   S708_TL_DC_U262_1_UP_DN.Error_T1.STATE := B#16#0;
   S708_TL_DC_U262_1_UP_DN.Error_T1.STIME := T#23D5H8M46S781MS;
   S708_TL_DC_U262_1_UP_DN.Error_T1.ATIME := T#23D5H8M46S825MS;
   S708_TL_DC_U262_1_UP_DN.Error_T2.IN := FALSE;
   S708_TL_DC_U262_1_UP_DN.Error_T2.PT := T#4S;
   S708_TL_DC_U262_1_UP_DN.Error_T2.Q := FALSE;
   S708_TL_DC_U262_1_UP_DN.Error_T2.ET := T#0MS;
   S708_TL_DC_U262_1_UP_DN.Error_T2.STATE := B#16#0;
   S708_TL_DC_U262_1_UP_DN.Error_T2.STIME := T#0MS;
   S708_TL_DC_U262_1_UP_DN.Error_T2.ATIME := T#0MS;
   S708_TL_DC_U262_1_UP_DN.Adv_End_Aux := FALSE;
   S708_TL_DC_U262_1_UP_DN.Ret_End_Aux := FALSE;
   S708_TL_DC_U262_1_UP_DN.CHK_Aux1 := FALSE;
   S708_TL_DC_U262_1_UP_DN.CHK_Aux2 := FALSE;
   S708_TL_DC_U262_1_UP_DN.Error_T1_DN := FALSE;
   S708_TL_DC_U262_1_UP_DN.Error_T2_DN := FALSE;
   S708_TL_DC_U262_1_UP_DN.Adv_Memo := FALSE;
   S708_TL_DC_U262_1_UP_DN.Visu_Adv_Arr[0] := FALSE;
   S708_TL_DC_U262_1_UP_DN.Visu_Adv_Arr[1] := FALSE;
   S708_TL_DC_U262_1_UP_DN.Visu_Adv_Arr[2] := FALSE;
   S708_TL_DC_U262_1_UP_DN.Visu_Adv_Arr[3] := FALSE;
   S708_TL_DC_U262_1_UP_DN.Visu_Adv_Arr[4] := FALSE;
   S708_TL_DC_U262_1_UP_DN.Visu_Adv_Arr[5] := FALSE;
   S708_TL_DC_U262_1_UP_DN.Visu_Adv_Arr[6] := FALSE;
   S708_TL_DC_U262_1_UP_DN.Visu_Adv_Arr[7] := FALSE;
   S708_TL_DC_U262_1_UP_DN.Visu_Adv_Arr[8] := FALSE;
   S708_TL_DC_U262_1_UP_DN.Visu_Adv_Arr[9] := FALSE;
   S708_TL_DC_U262_1_UP_DN.Visu_Adv_Arr[10] := FALSE;
   S708_TL_DC_U262_1_UP_DN.Visu_Adv_Arr[11] := FALSE;
   S708_TL_DC_U262_1_UP_DN.Visu_Adv_Arr[12] := FALSE;
   S708_TL_DC_U262_1_UP_DN.Visu_Adv_Arr[13] := FALSE;
   S708_TL_DC_U262_1_UP_DN.Visu_Adv_Arr[14] := FALSE;
   S708_TL_DC_U262_1_UP_DN.Visu_Adv_Arr[15] := FALSE;
   S708_TL_DC_U262_1_UP_DN.Visu_Ret_Arr[0] := FALSE;
   S708_TL_DC_U262_1_UP_DN.Visu_Ret_Arr[1] := FALSE;
   S708_TL_DC_U262_1_UP_DN.Visu_Ret_Arr[2] := FALSE;
   S708_TL_DC_U262_1_UP_DN.Visu_Ret_Arr[3] := FALSE;
   S708_TL_DC_U262_1_UP_DN.Visu_Ret_Arr[4] := FALSE;
   S708_TL_DC_U262_1_UP_DN.Visu_Ret_Arr[5] := FALSE;
   S708_TL_DC_U262_1_UP_DN.Visu_Ret_Arr[6] := FALSE;
   S708_TL_DC_U262_1_UP_DN.Visu_Ret_Arr[7] := FALSE;
   S708_TL_DC_U262_1_UP_DN.Visu_Ret_Arr[8] := FALSE;
   S708_TL_DC_U262_1_UP_DN.Visu_Ret_Arr[9] := FALSE;
   S708_TL_DC_U262_1_UP_DN.Visu_Ret_Arr[10] := FALSE;
   S708_TL_DC_U262_1_UP_DN.Visu_Ret_Arr[11] := FALSE;
   S708_TL_DC_U262_1_UP_DN.Visu_Ret_Arr[12] := FALSE;
   S708_TL_DC_U262_1_UP_DN.Visu_Ret_Arr[13] := FALSE;
   S708_TL_DC_U262_1_UP_DN.Visu_Ret_Arr[14] := FALSE;
   S708_TL_DC_U262_1_UP_DN.Visu_Ret_Arr[15] := FALSE;
   S708_TL_DC_U262_1_UP_DN.BLK_Move_Ret := 0;
   S708_TL_DC_U262_1_UP_DN.Enable := FALSE;
   S708_TL_DC_U262_1_UP_DN.Adv_End := FALSE;
   S708_TL_DC_U262_1_UP_DN.Ret_End := FALSE;
   S708_TL_DC_U262_1.Enable_Aux := FALSE;
   S708_TL_DC_U262_1.Adv_Amount := 1;
   S708_TL_DC_U262_1.Ret_Amount := 1;
   S708_TL_DC_U262_1.LS_Adv1 := FALSE;
   S708_TL_DC_U262_1.LS_Ret1 := FALSE;
   S708_TL_DC_U262_1.LS_Adv2 := FALSE;
   S708_TL_DC_U262_1.LS_Ret2 := FALSE;
   S708_TL_DC_U262_1.LS_Adv3 := FALSE;
   S708_TL_DC_U262_1.LS_Ret3 := FALSE;
   S708_TL_DC_U262_1.LS_Adv4 := FALSE;
   S708_TL_DC_U262_1.LS_Ret4 := FALSE;
   S708_TL_DC_U262_1.LS_Adv5 := FALSE;
   S708_TL_DC_U262_1.LS_Ret5 := FALSE;
   S708_TL_DC_U262_1.LS_Adv6 := FALSE;
   S708_TL_DC_U262_1.LS_Ret6 := FALSE;
   S708_TL_DC_U262_1.LS_Adv7 := FALSE;
   S708_TL_DC_U262_1.LS_Ret7 := FALSE;
   S708_TL_DC_U262_1.LS_Adv8 := FALSE;
   S708_TL_DC_U262_1.LS_Ret8 := FALSE;
   S708_TL_DC_U262_1.SOL_Adv := FALSE;
   S708_TL_DC_U262_1.SOL_Ret := FALSE;
   S708_TL_DC_U262_1.M_Ready := TRUE;
   S708_TL_DC_U262_1.T_CHK1 := T#4S;
   S708_TL_DC_U262_1.T_CHK2 := T#4S;
   S708_TL_DC_U262_1.PB_Lamp_CHK := FALSE;
   S708_TL_DC_U262_1.PB_Error_Rst := FALSE;
   S708_TL_DC_U262_1.M_FLICK := TRUE;
   S708_TL_DC_U262_1.M_Adv_Err := FALSE;
   S708_TL_DC_U262_1.M_Ret_Err := FALSE;
   S708_TL_DC_U262_1.LP_Adv := FALSE;
   S708_TL_DC_U262_1.LP_Ret := FALSE;
   S708_TL_DC_U262_1.Visu_Adv := W#16#0;
   S708_TL_DC_U262_1.Visu_Ret := W#16#0;
   S708_TL_DC_U262_1.Error_T1.IN := FALSE;
   S708_TL_DC_U262_1.Error_T1.PT := T#4S;
   S708_TL_DC_U262_1.Error_T1.Q := FALSE;
   S708_TL_DC_U262_1.Error_T1.ET := T#0MS;
   S708_TL_DC_U262_1.Error_T1.STATE := B#16#0;
   S708_TL_DC_U262_1.Error_T1.STIME := T#23D5H8M46S781MS;
   S708_TL_DC_U262_1.Error_T1.ATIME := T#23D5H8M46S825MS;
   S708_TL_DC_U262_1.Error_T2.IN := FALSE;
   S708_TL_DC_U262_1.Error_T2.PT := T#4S;
   S708_TL_DC_U262_1.Error_T2.Q := FALSE;
   S708_TL_DC_U262_1.Error_T2.ET := T#0MS;
   S708_TL_DC_U262_1.Error_T2.STATE := B#16#0;
   S708_TL_DC_U262_1.Error_T2.STIME := T#13H51M46S5MS;
   S708_TL_DC_U262_1.Error_T2.ATIME := T#13H51M46S50MS;
   S708_TL_DC_U262_1.Adv_End_Aux := FALSE;
   S708_TL_DC_U262_1.Ret_End_Aux := FALSE;
   S708_TL_DC_U262_1.CHK_Aux1 := FALSE;
   S708_TL_DC_U262_1.CHK_Aux2 := FALSE;
   S708_TL_DC_U262_1.Error_T1_DN := FALSE;
   S708_TL_DC_U262_1.Error_T2_DN := FALSE;
   S708_TL_DC_U262_1.Adv_Memo := FALSE;
   S708_TL_DC_U262_1.Visu_Adv_Arr[0] := FALSE;
   S708_TL_DC_U262_1.Visu_Adv_Arr[1] := FALSE;
   S708_TL_DC_U262_1.Visu_Adv_Arr[2] := FALSE;
   S708_TL_DC_U262_1.Visu_Adv_Arr[3] := FALSE;
   S708_TL_DC_U262_1.Visu_Adv_Arr[4] := FALSE;
   S708_TL_DC_U262_1.Visu_Adv_Arr[5] := FALSE;
   S708_TL_DC_U262_1.Visu_Adv_Arr[6] := FALSE;
   S708_TL_DC_U262_1.Visu_Adv_Arr[7] := FALSE;
   S708_TL_DC_U262_1.Visu_Adv_Arr[8] := FALSE;
   S708_TL_DC_U262_1.Visu_Adv_Arr[9] := FALSE;
   S708_TL_DC_U262_1.Visu_Adv_Arr[10] := FALSE;
   S708_TL_DC_U262_1.Visu_Adv_Arr[11] := FALSE;
   S708_TL_DC_U262_1.Visu_Adv_Arr[12] := FALSE;
   S708_TL_DC_U262_1.Visu_Adv_Arr[13] := FALSE;
   S708_TL_DC_U262_1.Visu_Adv_Arr[14] := FALSE;
   S708_TL_DC_U262_1.Visu_Adv_Arr[15] := FALSE;
   S708_TL_DC_U262_1.Visu_Ret_Arr[0] := FALSE;
   S708_TL_DC_U262_1.Visu_Ret_Arr[1] := FALSE;
   S708_TL_DC_U262_1.Visu_Ret_Arr[2] := FALSE;
   S708_TL_DC_U262_1.Visu_Ret_Arr[3] := FALSE;
   S708_TL_DC_U262_1.Visu_Ret_Arr[4] := FALSE;
   S708_TL_DC_U262_1.Visu_Ret_Arr[5] := FALSE;
   S708_TL_DC_U262_1.Visu_Ret_Arr[6] := FALSE;
   S708_TL_DC_U262_1.Visu_Ret_Arr[7] := FALSE;
   S708_TL_DC_U262_1.Visu_Ret_Arr[8] := FALSE;
   S708_TL_DC_U262_1.Visu_Ret_Arr[9] := FALSE;
   S708_TL_DC_U262_1.Visu_Ret_Arr[10] := FALSE;
   S708_TL_DC_U262_1.Visu_Ret_Arr[11] := FALSE;
   S708_TL_DC_U262_1.Visu_Ret_Arr[12] := FALSE;
   S708_TL_DC_U262_1.Visu_Ret_Arr[13] := FALSE;
   S708_TL_DC_U262_1.Visu_Ret_Arr[14] := FALSE;
   S708_TL_DC_U262_1.Visu_Ret_Arr[15] := FALSE;
   S708_TL_DC_U262_1.BLK_Move_Ret := 0;
   S708_TL_DC_U262_1.Enable := FALSE;
   S708_TL_DC_U262_1.Adv_End := FALSE;
   S708_TL_DC_U262_1.Ret_End := FALSE;
   S708_TL_DC_U262_1_CLAMP.Enable_Aux := FALSE;
   S708_TL_DC_U262_1_CLAMP.Adv_Amount := 1;
   S708_TL_DC_U262_1_CLAMP.Ret_Amount := 1;
   S708_TL_DC_U262_1_CLAMP.LS_Adv1 := FALSE;
   S708_TL_DC_U262_1_CLAMP.LS_Ret1 := FALSE;
   S708_TL_DC_U262_1_CLAMP.LS_Adv2 := FALSE;
   S708_TL_DC_U262_1_CLAMP.LS_Ret2 := FALSE;
   S708_TL_DC_U262_1_CLAMP.LS_Adv3 := FALSE;
   S708_TL_DC_U262_1_CLAMP.LS_Ret3 := FALSE;
   S708_TL_DC_U262_1_CLAMP.LS_Adv4 := FALSE;
   S708_TL_DC_U262_1_CLAMP.LS_Ret4 := FALSE;
   S708_TL_DC_U262_1_CLAMP.LS_Adv5 := FALSE;
   S708_TL_DC_U262_1_CLAMP.LS_Ret5 := FALSE;
   S708_TL_DC_U262_1_CLAMP.LS_Adv6 := FALSE;
   S708_TL_DC_U262_1_CLAMP.LS_Ret6 := FALSE;
   S708_TL_DC_U262_1_CLAMP.LS_Adv7 := FALSE;
   S708_TL_DC_U262_1_CLAMP.LS_Ret7 := FALSE;
   S708_TL_DC_U262_1_CLAMP.LS_Adv8 := FALSE;
   S708_TL_DC_U262_1_CLAMP.LS_Ret8 := FALSE;
   S708_TL_DC_U262_1_CLAMP.SOL_Adv := FALSE;
   S708_TL_DC_U262_1_CLAMP.SOL_Ret := FALSE;
   S708_TL_DC_U262_1_CLAMP.M_Ready := TRUE;
   S708_TL_DC_U262_1_CLAMP.T_CHK1 := T#4S;
   S708_TL_DC_U262_1_CLAMP.T_CHK2 := T#4S;
   S708_TL_DC_U262_1_CLAMP.PB_Lamp_CHK := FALSE;
   S708_TL_DC_U262_1_CLAMP.PB_Error_Rst := FALSE;
   S708_TL_DC_U262_1_CLAMP.M_FLICK := TRUE;
   S708_TL_DC_U262_1_CLAMP.M_Adv_Err := FALSE;
   S708_TL_DC_U262_1_CLAMP.M_Ret_Err := FALSE;
   S708_TL_DC_U262_1_CLAMP.LP_Adv := FALSE;
   S708_TL_DC_U262_1_CLAMP.LP_Ret := FALSE;
   S708_TL_DC_U262_1_CLAMP.Visu_Adv := W#16#0;
   S708_TL_DC_U262_1_CLAMP.Visu_Ret := W#16#0;
   S708_TL_DC_U262_1_CLAMP.Error_T1.IN := FALSE;
   S708_TL_DC_U262_1_CLAMP.Error_T1.PT := T#4S;
   S708_TL_DC_U262_1_CLAMP.Error_T1.Q := FALSE;
   S708_TL_DC_U262_1_CLAMP.Error_T1.ET := T#0MS;
   S708_TL_DC_U262_1_CLAMP.Error_T1.STATE := B#16#0;
   S708_TL_DC_U262_1_CLAMP.Error_T1.STIME := T#23D5H8M46S781MS;
   S708_TL_DC_U262_1_CLAMP.Error_T1.ATIME := T#23D5H8M46S825MS;
   S708_TL_DC_U262_1_CLAMP.Error_T2.IN := FALSE;
   S708_TL_DC_U262_1_CLAMP.Error_T2.PT := T#4S;
   S708_TL_DC_U262_1_CLAMP.Error_T2.Q := FALSE;
   S708_TL_DC_U262_1_CLAMP.Error_T2.ET := T#0MS;
   S708_TL_DC_U262_1_CLAMP.Error_T2.STATE := B#16#0;
   S708_TL_DC_U262_1_CLAMP.Error_T2.STIME := T#0MS;
   S708_TL_DC_U262_1_CLAMP.Error_T2.ATIME := T#0MS;
   S708_TL_DC_U262_1_CLAMP.Adv_End_Aux := FALSE;
   S708_TL_DC_U262_1_CLAMP.Ret_End_Aux := FALSE;
   S708_TL_DC_U262_1_CLAMP.CHK_Aux1 := FALSE;
   S708_TL_DC_U262_1_CLAMP.CHK_Aux2 := FALSE;
   S708_TL_DC_U262_1_CLAMP.Error_T1_DN := FALSE;
   S708_TL_DC_U262_1_CLAMP.Error_T2_DN := FALSE;
   S708_TL_DC_U262_1_CLAMP.Adv_Memo := FALSE;
   S708_TL_DC_U262_1_CLAMP.Visu_Adv_Arr[0] := FALSE;
   S708_TL_DC_U262_1_CLAMP.Visu_Adv_Arr[1] := FALSE;
   S708_TL_DC_U262_1_CLAMP.Visu_Adv_Arr[2] := FALSE;
   S708_TL_DC_U262_1_CLAMP.Visu_Adv_Arr[3] := FALSE;
   S708_TL_DC_U262_1_CLAMP.Visu_Adv_Arr[4] := FALSE;
   S708_TL_DC_U262_1_CLAMP.Visu_Adv_Arr[5] := FALSE;
   S708_TL_DC_U262_1_CLAMP.Visu_Adv_Arr[6] := FALSE;
   S708_TL_DC_U262_1_CLAMP.Visu_Adv_Arr[7] := FALSE;
   S708_TL_DC_U262_1_CLAMP.Visu_Adv_Arr[8] := FALSE;
   S708_TL_DC_U262_1_CLAMP.Visu_Adv_Arr[9] := FALSE;
   S708_TL_DC_U262_1_CLAMP.Visu_Adv_Arr[10] := FALSE;
   S708_TL_DC_U262_1_CLAMP.Visu_Adv_Arr[11] := FALSE;
   S708_TL_DC_U262_1_CLAMP.Visu_Adv_Arr[12] := FALSE;
   S708_TL_DC_U262_1_CLAMP.Visu_Adv_Arr[13] := FALSE;
   S708_TL_DC_U262_1_CLAMP.Visu_Adv_Arr[14] := FALSE;
   S708_TL_DC_U262_1_CLAMP.Visu_Adv_Arr[15] := FALSE;
   S708_TL_DC_U262_1_CLAMP.Visu_Ret_Arr[0] := FALSE;
   S708_TL_DC_U262_1_CLAMP.Visu_Ret_Arr[1] := FALSE;
   S708_TL_DC_U262_1_CLAMP.Visu_Ret_Arr[2] := FALSE;
   S708_TL_DC_U262_1_CLAMP.Visu_Ret_Arr[3] := FALSE;
   S708_TL_DC_U262_1_CLAMP.Visu_Ret_Arr[4] := FALSE;
   S708_TL_DC_U262_1_CLAMP.Visu_Ret_Arr[5] := FALSE;
   S708_TL_DC_U262_1_CLAMP.Visu_Ret_Arr[6] := FALSE;
   S708_TL_DC_U262_1_CLAMP.Visu_Ret_Arr[7] := FALSE;
   S708_TL_DC_U262_1_CLAMP.Visu_Ret_Arr[8] := FALSE;
   S708_TL_DC_U262_1_CLAMP.Visu_Ret_Arr[9] := FALSE;
   S708_TL_DC_U262_1_CLAMP.Visu_Ret_Arr[10] := FALSE;
   S708_TL_DC_U262_1_CLAMP.Visu_Ret_Arr[11] := FALSE;
   S708_TL_DC_U262_1_CLAMP.Visu_Ret_Arr[12] := FALSE;
   S708_TL_DC_U262_1_CLAMP.Visu_Ret_Arr[13] := FALSE;
   S708_TL_DC_U262_1_CLAMP.Visu_Ret_Arr[14] := FALSE;
   S708_TL_DC_U262_1_CLAMP.Visu_Ret_Arr[15] := FALSE;
   S708_TL_DC_U262_1_CLAMP.BLK_Move_Ret := 0;
   S708_TL_DC_U262_1_CLAMP.Enable := FALSE;
   S708_TL_DC_U262_1_CLAMP.Adv_End := FALSE;
   S708_TL_DC_U262_1_CLAMP.Ret_End := FALSE;
   S708_TL_DC_U261_2_CLAMP.Enable_Aux := FALSE;
   S708_TL_DC_U261_2_CLAMP.Adv_Amount := 1;
   S708_TL_DC_U261_2_CLAMP.Ret_Amount := 1;
   S708_TL_DC_U261_2_CLAMP.LS_Adv1 := FALSE;
   S708_TL_DC_U261_2_CLAMP.LS_Ret1 := FALSE;
   S708_TL_DC_U261_2_CLAMP.LS_Adv2 := FALSE;
   S708_TL_DC_U261_2_CLAMP.LS_Ret2 := FALSE;
   S708_TL_DC_U261_2_CLAMP.LS_Adv3 := FALSE;
   S708_TL_DC_U261_2_CLAMP.LS_Ret3 := FALSE;
   S708_TL_DC_U261_2_CLAMP.LS_Adv4 := FALSE;
   S708_TL_DC_U261_2_CLAMP.LS_Ret4 := FALSE;
   S708_TL_DC_U261_2_CLAMP.LS_Adv5 := FALSE;
   S708_TL_DC_U261_2_CLAMP.LS_Ret5 := FALSE;
   S708_TL_DC_U261_2_CLAMP.LS_Adv6 := FALSE;
   S708_TL_DC_U261_2_CLAMP.LS_Ret6 := FALSE;
   S708_TL_DC_U261_2_CLAMP.LS_Adv7 := FALSE;
   S708_TL_DC_U261_2_CLAMP.LS_Ret7 := FALSE;
   S708_TL_DC_U261_2_CLAMP.LS_Adv8 := FALSE;
   S708_TL_DC_U261_2_CLAMP.LS_Ret8 := FALSE;
   S708_TL_DC_U261_2_CLAMP.SOL_Adv := FALSE;
   S708_TL_DC_U261_2_CLAMP.SOL_Ret := FALSE;
   S708_TL_DC_U261_2_CLAMP.M_Ready := TRUE;
   S708_TL_DC_U261_2_CLAMP.T_CHK1 := T#4S;
   S708_TL_DC_U261_2_CLAMP.T_CHK2 := T#4S;
   S708_TL_DC_U261_2_CLAMP.PB_Lamp_CHK := FALSE;
   S708_TL_DC_U261_2_CLAMP.PB_Error_Rst := FALSE;
   S708_TL_DC_U261_2_CLAMP.M_FLICK := TRUE;
   S708_TL_DC_U261_2_CLAMP.M_Adv_Err := FALSE;
   S708_TL_DC_U261_2_CLAMP.M_Ret_Err := FALSE;
   S708_TL_DC_U261_2_CLAMP.LP_Adv := FALSE;
   S708_TL_DC_U261_2_CLAMP.LP_Ret := FALSE;
   S708_TL_DC_U261_2_CLAMP.Visu_Adv := W#16#0;
   S708_TL_DC_U261_2_CLAMP.Visu_Ret := W#16#0;
   S708_TL_DC_U261_2_CLAMP.Error_T1.IN := FALSE;
   S708_TL_DC_U261_2_CLAMP.Error_T1.PT := T#4S;
   S708_TL_DC_U261_2_CLAMP.Error_T1.Q := FALSE;
   S708_TL_DC_U261_2_CLAMP.Error_T1.ET := T#0MS;
   S708_TL_DC_U261_2_CLAMP.Error_T1.STATE := B#16#0;
   S708_TL_DC_U261_2_CLAMP.Error_T1.STIME := T#23D5H8M46S781MS;
   S708_TL_DC_U261_2_CLAMP.Error_T1.ATIME := T#23D5H8M46S825MS;
   S708_TL_DC_U261_2_CLAMP.Error_T2.IN := FALSE;
   S708_TL_DC_U261_2_CLAMP.Error_T2.PT := T#4S;
   S708_TL_DC_U261_2_CLAMP.Error_T2.Q := FALSE;
   S708_TL_DC_U261_2_CLAMP.Error_T2.ET := T#0MS;
   S708_TL_DC_U261_2_CLAMP.Error_T2.STATE := B#16#0;
   S708_TL_DC_U261_2_CLAMP.Error_T2.STIME := T#0MS;
   S708_TL_DC_U261_2_CLAMP.Error_T2.ATIME := T#0MS;
   S708_TL_DC_U261_2_CLAMP.Adv_End_Aux := FALSE;
   S708_TL_DC_U261_2_CLAMP.Ret_End_Aux := FALSE;
   S708_TL_DC_U261_2_CLAMP.CHK_Aux1 := FALSE;
   S708_TL_DC_U261_2_CLAMP.CHK_Aux2 := FALSE;
   S708_TL_DC_U261_2_CLAMP.Error_T1_DN := FALSE;
   S708_TL_DC_U261_2_CLAMP.Error_T2_DN := FALSE;
   S708_TL_DC_U261_2_CLAMP.Adv_Memo := FALSE;
   S708_TL_DC_U261_2_CLAMP.Visu_Adv_Arr[0] := FALSE;
   S708_TL_DC_U261_2_CLAMP.Visu_Adv_Arr[1] := FALSE;
   S708_TL_DC_U261_2_CLAMP.Visu_Adv_Arr[2] := FALSE;
   S708_TL_DC_U261_2_CLAMP.Visu_Adv_Arr[3] := FALSE;
   S708_TL_DC_U261_2_CLAMP.Visu_Adv_Arr[4] := FALSE;
   S708_TL_DC_U261_2_CLAMP.Visu_Adv_Arr[5] := FALSE;
   S708_TL_DC_U261_2_CLAMP.Visu_Adv_Arr[6] := FALSE;
   S708_TL_DC_U261_2_CLAMP.Visu_Adv_Arr[7] := FALSE;
   S708_TL_DC_U261_2_CLAMP.Visu_Adv_Arr[8] := FALSE;
   S708_TL_DC_U261_2_CLAMP.Visu_Adv_Arr[9] := FALSE;
   S708_TL_DC_U261_2_CLAMP.Visu_Adv_Arr[10] := FALSE;
   S708_TL_DC_U261_2_CLAMP.Visu_Adv_Arr[11] := FALSE;
   S708_TL_DC_U261_2_CLAMP.Visu_Adv_Arr[12] := FALSE;
   S708_TL_DC_U261_2_CLAMP.Visu_Adv_Arr[13] := FALSE;
   S708_TL_DC_U261_2_CLAMP.Visu_Adv_Arr[14] := FALSE;
   S708_TL_DC_U261_2_CLAMP.Visu_Adv_Arr[15] := FALSE;
   S708_TL_DC_U261_2_CLAMP.Visu_Ret_Arr[0] := FALSE;
   S708_TL_DC_U261_2_CLAMP.Visu_Ret_Arr[1] := FALSE;
   S708_TL_DC_U261_2_CLAMP.Visu_Ret_Arr[2] := FALSE;
   S708_TL_DC_U261_2_CLAMP.Visu_Ret_Arr[3] := FALSE;
   S708_TL_DC_U261_2_CLAMP.Visu_Ret_Arr[4] := FALSE;
   S708_TL_DC_U261_2_CLAMP.Visu_Ret_Arr[5] := FALSE;
   S708_TL_DC_U261_2_CLAMP.Visu_Ret_Arr[6] := FALSE;
   S708_TL_DC_U261_2_CLAMP.Visu_Ret_Arr[7] := FALSE;
   S708_TL_DC_U261_2_CLAMP.Visu_Ret_Arr[8] := FALSE;
   S708_TL_DC_U261_2_CLAMP.Visu_Ret_Arr[9] := FALSE;
   S708_TL_DC_U261_2_CLAMP.Visu_Ret_Arr[10] := FALSE;
   S708_TL_DC_U261_2_CLAMP.Visu_Ret_Arr[11] := FALSE;
   S708_TL_DC_U261_2_CLAMP.Visu_Ret_Arr[12] := FALSE;
   S708_TL_DC_U261_2_CLAMP.Visu_Ret_Arr[13] := FALSE;
   S708_TL_DC_U261_2_CLAMP.Visu_Ret_Arr[14] := FALSE;
   S708_TL_DC_U261_2_CLAMP.Visu_Ret_Arr[15] := FALSE;
   S708_TL_DC_U261_2_CLAMP.BLK_Move_Ret := 0;
   S708_TL_DC_U261_2_CLAMP.Enable := FALSE;
   S708_TL_DC_U261_2_CLAMP.Adv_End := FALSE;
   S708_TL_DC_U261_2_CLAMP.Ret_End := FALSE;
END_DATA_BLOCK

FUNCTION FC 144 : VOID
TITLE =
VERSION : 0.1

BEGIN
NETWORK
TITLE =
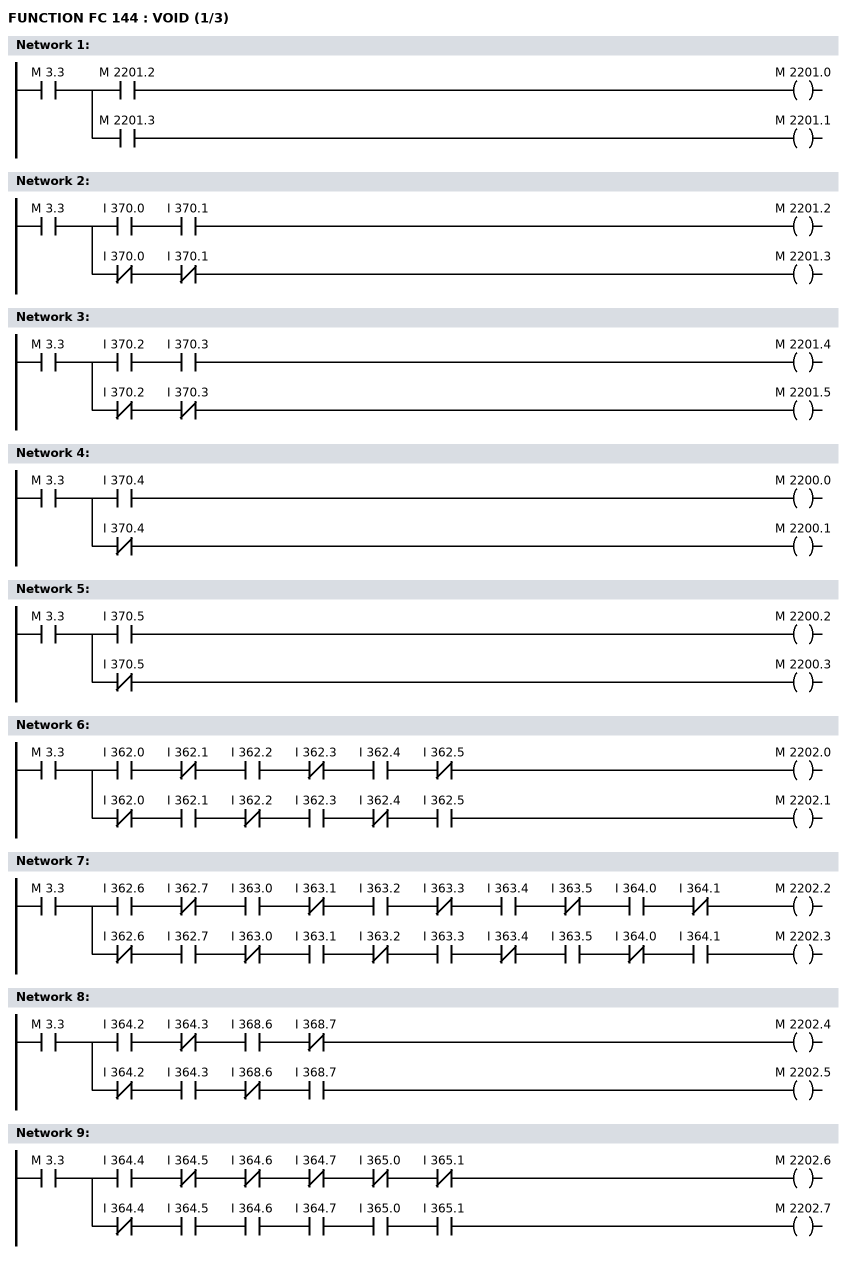

      A     M      3.3;
      =     L      0.0;
      A     L      0.0;
      A     M   2201.2;
      =     M   2201.0;
      A     L      0.0;
      A     M   2201.3;
      =     M   2201.1;
NETWORK
TITLE =

      A     M      3.3;
      =     L      0.0;
      A     L      0.0;
      A     I    370.0;
      A     I    370.1;
      =     M   2201.2;
      A     L      0.0;
      AN    I    370.0;
      AN    I    370.1;
      =     M   2201.3;
NETWORK
TITLE =

      A     M      3.3;
      =     L      0.0;
      A     L      0.0;
      A     I    370.2;
      A     I    370.3;
      =     M   2201.4;
      A     L      0.0;
      AN    I    370.2;
      AN    I    370.3;
      =     M   2201.5;
NETWORK
TITLE =

      A     M      3.3;
      =     L      0.0;
      A     L      0.0;
      A     I    370.4;
      =     M   2200.0;
      A     L      0.0;
      AN    I    370.4;
      =     M   2200.1;
NETWORK
TITLE =

      A     M      3.3;
      =     L      0.0;
      A     L      0.0;
      A     I    370.5;
      =     M   2200.2;
      A     L      0.0;
      AN    I    370.5;
      =     M   2200.3;
NETWORK
TITLE =

      A     M      3.3;
      =     L      0.0;
      A     L      0.0;
      A     I    362.0;
      AN    I    362.1;
      A     I    362.2;
      AN    I    362.3;
      A     I    362.4;
      AN    I    362.5;
      =     M   2202.0;
      A     L      0.0;
      AN    I    362.0;
      A     I    362.1;
      AN    I    362.2;
      A     I    362.3;
      AN    I    362.4;
      A     I    362.5;
      =     M   2202.1;
NETWORK
TITLE =

      A     M      3.3;
      =     L      0.0;
      A     L      0.0;
      A     I    362.6;
      AN    I    362.7;
      A     I    363.0;
      AN    I    363.1;
      A     I    363.2;
      AN    I    363.3;
      A     I    363.4;
      AN    I    363.5;
      A     I    364.0;
      AN    I    364.1;
      =     M   2202.2;
      A     L      0.0;
      AN    I    362.6;
      A     I    362.7;
      AN    I    363.0;
      A     I    363.1;
      AN    I    363.2;
      A     I    363.3;
      AN    I    363.4;
      A     I    363.5;
      AN    I    364.0;
      A     I    364.1;
      =     M   2202.3;
NETWORK
TITLE =

      A     M      3.3;
      =     L      0.0;
      A     L      0.0;
      A     I    364.2;
      AN    I    364.3;
      A     I    368.6;
      AN    I    368.7;
      =     M   2202.4;
      A     L      0.0;
      AN    I    364.2;
      A     I    364.3;
      AN    I    368.6;
      A     I    368.7;
      =     M   2202.5;
NETWORK
TITLE =

      A     M      3.3;
      =     L      0.0;
      A     L      0.0;
      A     I    364.4;
      AN    I    364.5;
      AN    I    364.6;
      AN    I    364.7;
      AN    I    365.0;
      AN    I    365.1;
      =     M   2202.6;
      A     L      0.0;
      AN    I    364.4;
      A     I    364.5;
      A     I    364.6;
      A     I    364.7;
      A     I    365.0;
      A     I    365.1;
      =     M   2202.7;
NETWORK
TITLE =
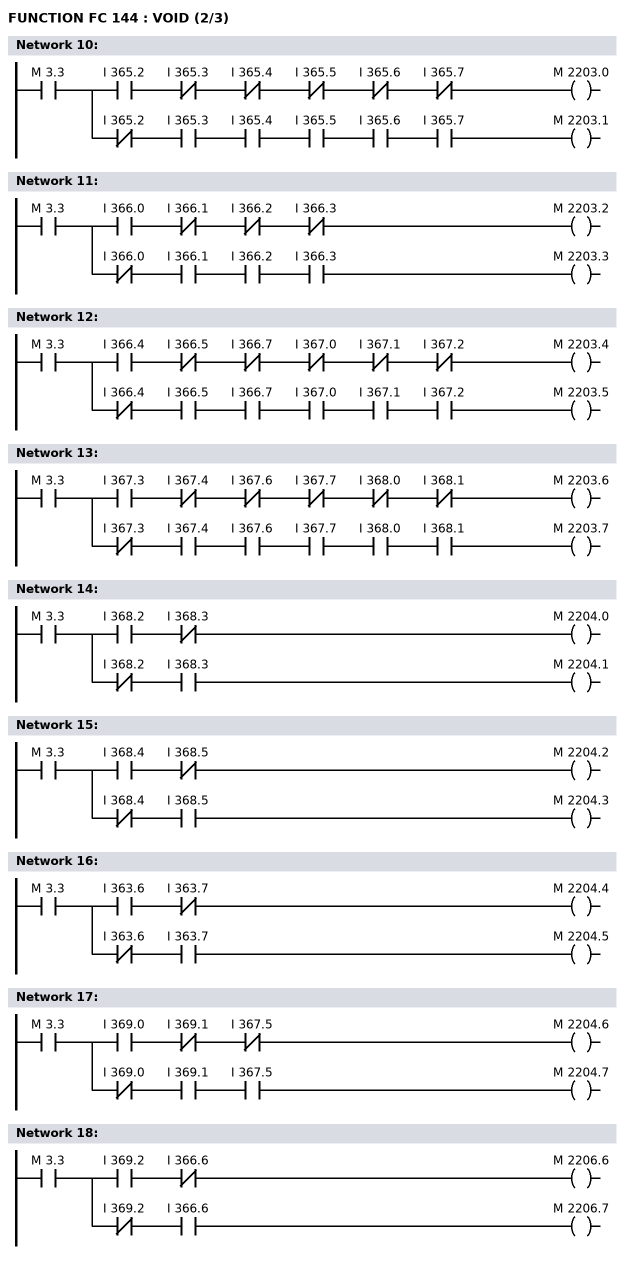

      A     M      3.3;
      =     L      0.0;
      A     L      0.0;
      A     I    365.2;
      AN    I    365.3;
      AN    I    365.4;
      AN    I    365.5;
      AN    I    365.6;
      AN    I    365.7;
      =     M   2203.0;
      A     L      0.0;
      AN    I    365.2;
      A     I    365.3;
      A     I    365.4;
      A     I    365.5;
      A     I    365.6;
      A     I    365.7;
      =     M   2203.1;
NETWORK
TITLE =

      A     M      3.3;
      =     L      0.0;
      A     L      0.0;
      A     I    366.0;
      AN    I    366.1;
      AN    I    366.2;
      AN    I    366.3;
      =     M   2203.2;
      A     L      0.0;
      AN    I    366.0;
      A     I    366.1;
      A     I    366.2;
      A     I    366.3;
      =     M   2203.3;
NETWORK
TITLE =

      A     M      3.3;
      =     L      0.0;
      A     L      0.0;
      A     I    366.4;
      AN    I    366.5;
      AN    I    366.7;
      AN    I    367.0;
      AN    I    367.1;
      AN    I    367.2;
      =     M   2203.4;
      A     L      0.0;
      AN    I    366.4;
      A     I    366.5;
      A     I    366.7;
      A     I    367.0;
      A     I    367.1;
      A     I    367.2;
      =     M   2203.5;
NETWORK
TITLE =

      A     M      3.3;
      =     L      0.0;
      A     L      0.0;
      A     I    367.3;
      AN    I    367.4;
      AN    I    367.6;
      AN    I    367.7;
      AN    I    368.0;
      AN    I    368.1;
      =     M   2203.6;
      A     L      0.0;
      AN    I    367.3;
      A     I    367.4;
      A     I    367.6;
      A     I    367.7;
      A     I    368.0;
      A     I    368.1;
      =     M   2203.7;
NETWORK
TITLE =

      A     M      3.3;
      =     L      0.0;
      A     L      0.0;
      A     I    368.2;
      AN    I    368.3;
      =     M   2204.0;
      A     L      0.0;
      AN    I    368.2;
      A     I    368.3;
      =     M   2204.1;
NETWORK
TITLE =

      A     M      3.3;
      =     L      0.0;
      A     L      0.0;
      A     I    368.4;
      AN    I    368.5;
      =     M   2204.2;
      A     L      0.0;
      AN    I    368.4;
      A     I    368.5;
      =     M   2204.3;
NETWORK
TITLE =

      A     M      3.3;
      =     L      0.0;
      A     L      0.0;
      A     I    363.6;
      AN    I    363.7;
      =     M   2204.4;
      A     L      0.0;
      AN    I    363.6;
      A     I    363.7;
      =     M   2204.5;
NETWORK
TITLE =

      A     M      3.3;
      =     L      0.0;
      A     L      0.0;
      A     I    369.0;
      AN    I    369.1;
      AN    I    367.5;
      =     M   2204.6;
      A     L      0.0;
      AN    I    369.0;
      A     I    369.1;
      A     I    367.5;
      =     M   2204.7;
NETWORK
TITLE =

      A     M      3.3;
      =     L      0.0;
      A     L      0.0;
      A     I    369.2;
      AN    I    366.6;
      =     M   2206.6;
      A     L      0.0;
      AN    I    369.2;
      A     I    366.6;
      =     M   2206.7;
NETWORK
TITLE =
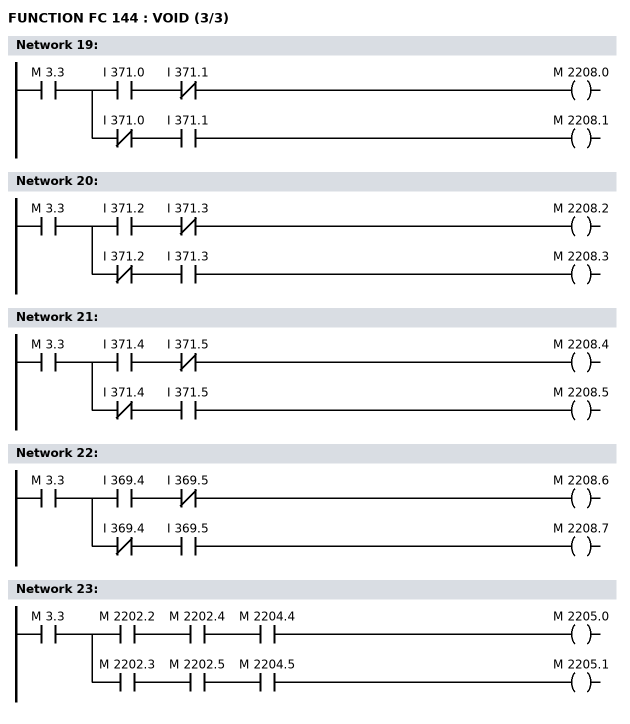

      A     M      3.3;
      =     L      0.0;
      A     L      0.0;
      A     I    371.0;
      AN    I    371.1;
      =     M   2208.0;
      A     L      0.0;
      AN    I    371.0;
      A     I    371.1;
      =     M   2208.1;
NETWORK
TITLE =

      A     M      3.3;
      =     L      0.0;
      A     L      0.0;
      A     I    371.2;
      AN    I    371.3;
      =     M   2208.2;
      A     L      0.0;
      AN    I    371.2;
      A     I    371.3;
      =     M   2208.3;
NETWORK
TITLE =

      A     M      3.3;
      =     L      0.0;
      A     L      0.0;
      A     I    371.4;
      AN    I    371.5;
      =     M   2208.4;
      A     L      0.0;
      AN    I    371.4;
      A     I    371.5;
      =     M   2208.5;
NETWORK
TITLE =

      A     M      3.3;
      =     L      0.0;
      A     L      0.0;
      A     I    369.4;
      AN    I    369.5;
      =     M   2208.6;
      A     L      0.0;
      AN    I    369.4;
      A     I    369.5;
      =     M   2208.7;
NETWORK
TITLE =

      A     M      3.3;
      =     L      0.0;
      A     L      0.0;
      A     M   2202.2;
      A     M   2202.4;
      A     M   2204.4;
      =     M   2205.0;
      A     L      0.0;
      A     M   2202.3;
      A     M   2202.5;
      A     M   2204.5;
      =     M   2205.1;
NETWORK
TITLE =

      A     M      3.3;
      =     L      0.0;
      A     L      0.0;
      A     M   2202.6;
      A     M   2203.0;
      A     M   2203.2;
      A     M   2203.4;
      A     M   2203.6;
      A     M   2206.6;
      =     L      0.1;
      A     L      0.1;
      BLD   102;
      =     M   2205.2;
      A     L      0.1;
      A     M   2204.2;
      A     M   2204.6;
      =     M   2205.4;
      A     L      0.0;
      A     M   2202.7;
      A     M   2203.1;
      A     M   2203.3;
      A     M   2203.5;
      A     M   2203.7;
      A     M   2206.7;
      =     L      0.1;
      A     L      0.1;
      BLD   102;
      =     M   2205.3;
      A     L      0.1;
      A     M   2204.3;
      A     M   2204.7;
      =     M   2205.5;
NETWORK
TITLE =
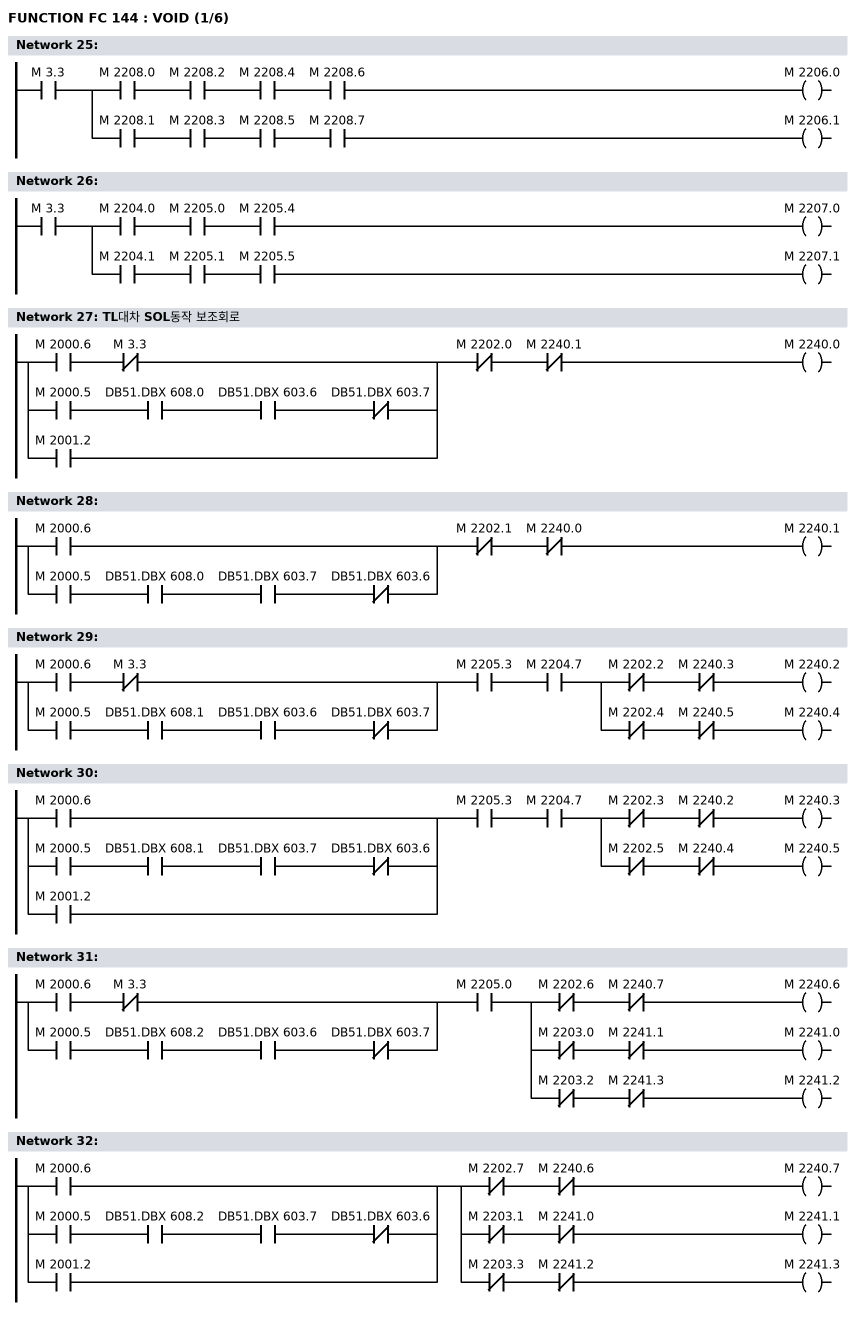

      A     M      3.3;
      =     L      0.0;
      A     L      0.0;
      A     M   2208.0;
      A     M   2208.2;
      A     M   2208.4;
      A     M   2208.6;
      =     M   2206.0;
      A     L      0.0;
      A     M   2208.1;
      A     M   2208.3;
      A     M   2208.5;
      A     M   2208.7;
      =     M   2206.1;
NETWORK
TITLE =

      A     M      3.3;
      =     L      0.0;
      A     L      0.0;
      A     M   2204.0;
      A     M   2205.0;
      A     M   2205.4;
      =     M   2207.0;
      A     L      0.0;
      A     M   2204.1;
      A     M   2205.1;
      A     M   2205.5;
      =     M   2207.1;
NETWORK
TITLE =TL대차 SOL동작 보조회로

      A(    ;
      A     M   2000.6;
      AN    M      3.3;
      O     ;
      A     M   2000.5;
      A     DB51.DBX  608.0;
      A     DB51.DBX  603.6;
      AN    DB51.DBX  603.7;
      O     M   2001.2;
      )     ;
      AN    M   2202.0;
      AN    M   2240.1;
      =     M   2240.0;
NETWORK
TITLE =

      A(    ;
      O     M   2000.6;
      O     ;
      A     M   2000.5;
      A     DB51.DBX  608.0;
      A     DB51.DBX  603.7;
      AN    DB51.DBX  603.6;
      )     ;
      AN    M   2202.1;
      AN    M   2240.0;
      =     M   2240.1;
NETWORK
TITLE =

      A(    ;
      A     M   2000.6;
      AN    M      3.3;
      O     ;
      A     M   2000.5;
      A     DB51.DBX  608.1;
      A     DB51.DBX  603.6;
      AN    DB51.DBX  603.7;
      )     ;
      A     M   2205.3;
      A     M   2204.7;
      =     L      0.0;
      A     L      0.0;
      AN    M   2202.2;
      AN    M   2240.3;
      =     M   2240.2;
      A     L      0.0;
      AN    M   2202.4;
      AN    M   2240.5;
      =     M   2240.4;
NETWORK
TITLE =

      A(    ;
      O     M   2000.6;
      O     ;
      A     M   2000.5;
      A     DB51.DBX  608.1;
      A     DB51.DBX  603.7;
      AN    DB51.DBX  603.6;
      O     M   2001.2;
      )     ;
      A     M   2205.3;
      A     M   2204.7;
      =     L      0.0;
      A     L      0.0;
      AN    M   2202.3;
      AN    M   2240.2;
      =     M   2240.3;
      A     L      0.0;
      AN    M   2202.5;
      AN    M   2240.4;
      =     M   2240.5;
NETWORK
TITLE =

      A(    ;
      A     M   2000.6;
      AN    M      3.3;
      O     ;
      A     M   2000.5;
      A     DB51.DBX  608.2;
      A     DB51.DBX  603.6;
      AN    DB51.DBX  603.7;
      )     ;
      A     M   2205.0;
      =     L      0.0;
      A     L      0.0;
      AN    M   2202.6;
      AN    M   2240.7;
      =     M   2240.6;
      A     L      0.0;
      AN    M   2203.0;
      AN    M   2241.1;
      =     M   2241.0;
      A     L      0.0;
      AN    M   2203.2;
      AN    M   2241.3;
      =     M   2241.2;
NETWORK
TITLE =

      O     M   2000.6;
      O     ;
      A     M   2000.5;
      A     DB51.DBX  608.2;
      A     DB51.DBX  603.7;
      AN    DB51.DBX  603.6;
      O     M   2001.2;
      =     L      0.0;
      A     L      0.0;
      AN    M   2202.7;
      AN    M   2240.6;
      =     M   2240.7;
      A     L      0.0;
      AN    M   2203.1;
      AN    M   2241.0;
      =     M   2241.1;
      A     L      0.0;
      AN    M   2203.3;
      AN    M   2241.2;
      =     M   2241.3;
NETWORK
TITLE =
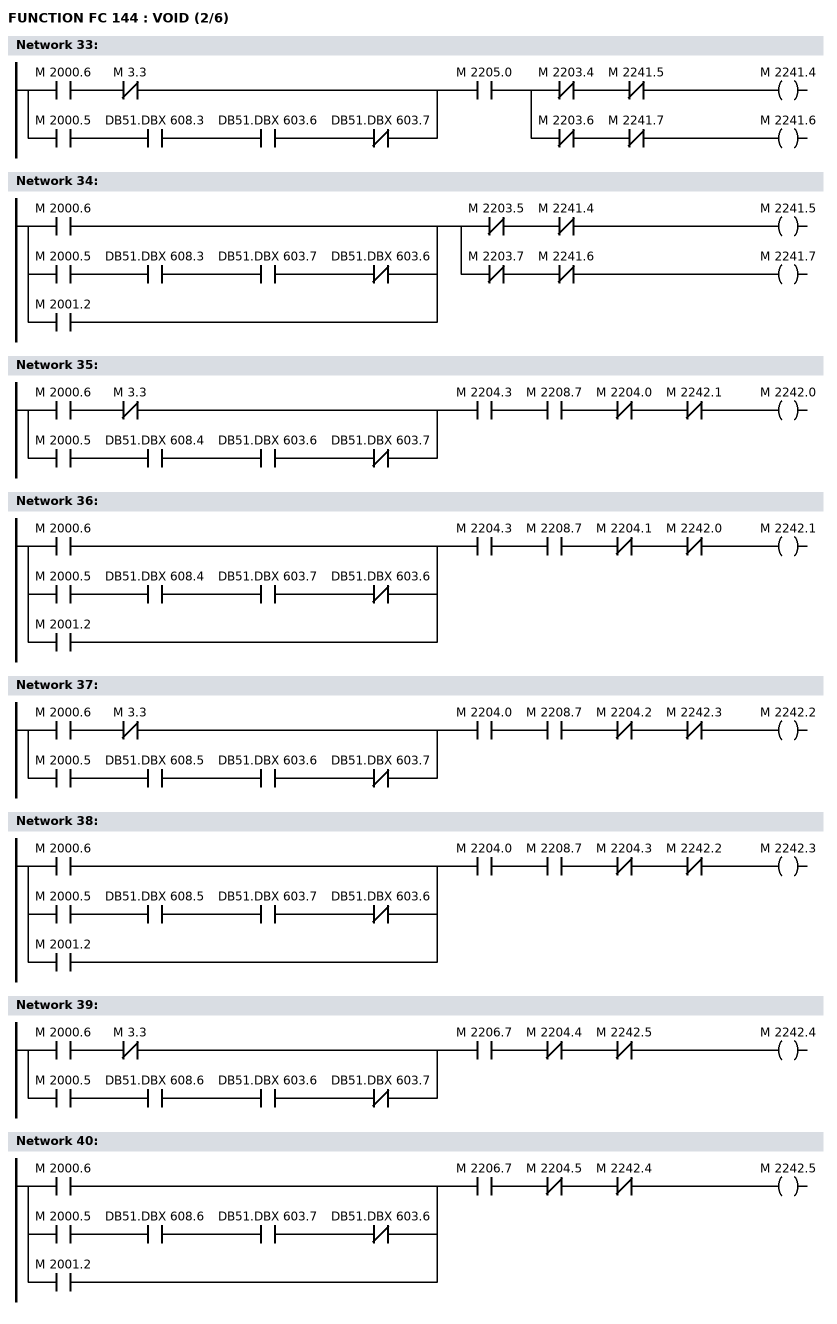

      A(    ;
      A     M   2000.6;
      AN    M      3.3;
      O     ;
      A     M   2000.5;
      A     DB51.DBX  608.3;
      A     DB51.DBX  603.6;
      AN    DB51.DBX  603.7;
      )     ;
      A     M   2205.0;
      =     L      0.0;
      A     L      0.0;
      AN    M   2203.4;
      AN    M   2241.5;
      =     M   2241.4;
      A     L      0.0;
      AN    M   2203.6;
      AN    M   2241.7;
      =     M   2241.6;
NETWORK
TITLE =

      O     M   2000.6;
      O     ;
      A     M   2000.5;
      A     DB51.DBX  608.3;
      A     DB51.DBX  603.7;
      AN    DB51.DBX  603.6;
      O     M   2001.2;
      =     L      0.0;
      A     L      0.0;
      AN    M   2203.5;
      AN    M   2241.4;
      =     M   2241.5;
      A     L      0.0;
      AN    M   2203.7;
      AN    M   2241.6;
      =     M   2241.7;
NETWORK
TITLE =

      A(    ;
      A     M   2000.6;
      AN    M      3.3;
      O     ;
      A     M   2000.5;
      A     DB51.DBX  608.4;
      A     DB51.DBX  603.6;
      AN    DB51.DBX  603.7;
      )     ;
      A     M   2204.3;
      A     M   2208.7;
      AN    M   2204.0;
      AN    M   2242.1;
      =     M   2242.0;
NETWORK
TITLE =

      A(    ;
      O     M   2000.6;
      O     ;
      A     M   2000.5;
      A     DB51.DBX  608.4;
      A     DB51.DBX  603.7;
      AN    DB51.DBX  603.6;
      O     M   2001.2;
      )     ;
      A     M   2204.3;
      A     M   2208.7;
      AN    M   2204.1;
      AN    M   2242.0;
      =     M   2242.1;
NETWORK
TITLE =

      A(    ;
      A     M   2000.6;
      AN    M      3.3;
      O     ;
      A     M   2000.5;
      A     DB51.DBX  608.5;
      A     DB51.DBX  603.6;
      AN    DB51.DBX  603.7;
      )     ;
      A     M   2204.0;
      A     M   2208.7;
      AN    M   2204.2;
      AN    M   2242.3;
      =     M   2242.2;
NETWORK
TITLE =

      A(    ;
      O     M   2000.6;
      O     ;
      A     M   2000.5;
      A     DB51.DBX  608.5;
      A     DB51.DBX  603.7;
      AN    DB51.DBX  603.6;
      O     M   2001.2;
      )     ;
      A     M   2204.0;
      A     M   2208.7;
      AN    M   2204.3;
      AN    M   2242.2;
      =     M   2242.3;
NETWORK
TITLE =

      A(    ;
      A     M   2000.6;
      AN    M      3.3;
      O     ;
      A     M   2000.5;
      A     DB51.DBX  608.6;
      A     DB51.DBX  603.6;
      AN    DB51.DBX  603.7;
      )     ;
      A     M   2206.7;
      AN    M   2204.4;
      AN    M   2242.5;
      =     M   2242.4;
NETWORK
TITLE =

      A(    ;
      O     M   2000.6;
      O     ;
      A     M   2000.5;
      A     DB51.DBX  608.6;
      A     DB51.DBX  603.7;
      AN    DB51.DBX  603.6;
      O     M   2001.2;
      )     ;
      A     M   2206.7;
      AN    M   2204.5;
      AN    M   2242.4;
      =     M   2242.5;
NETWORK
TITLE =
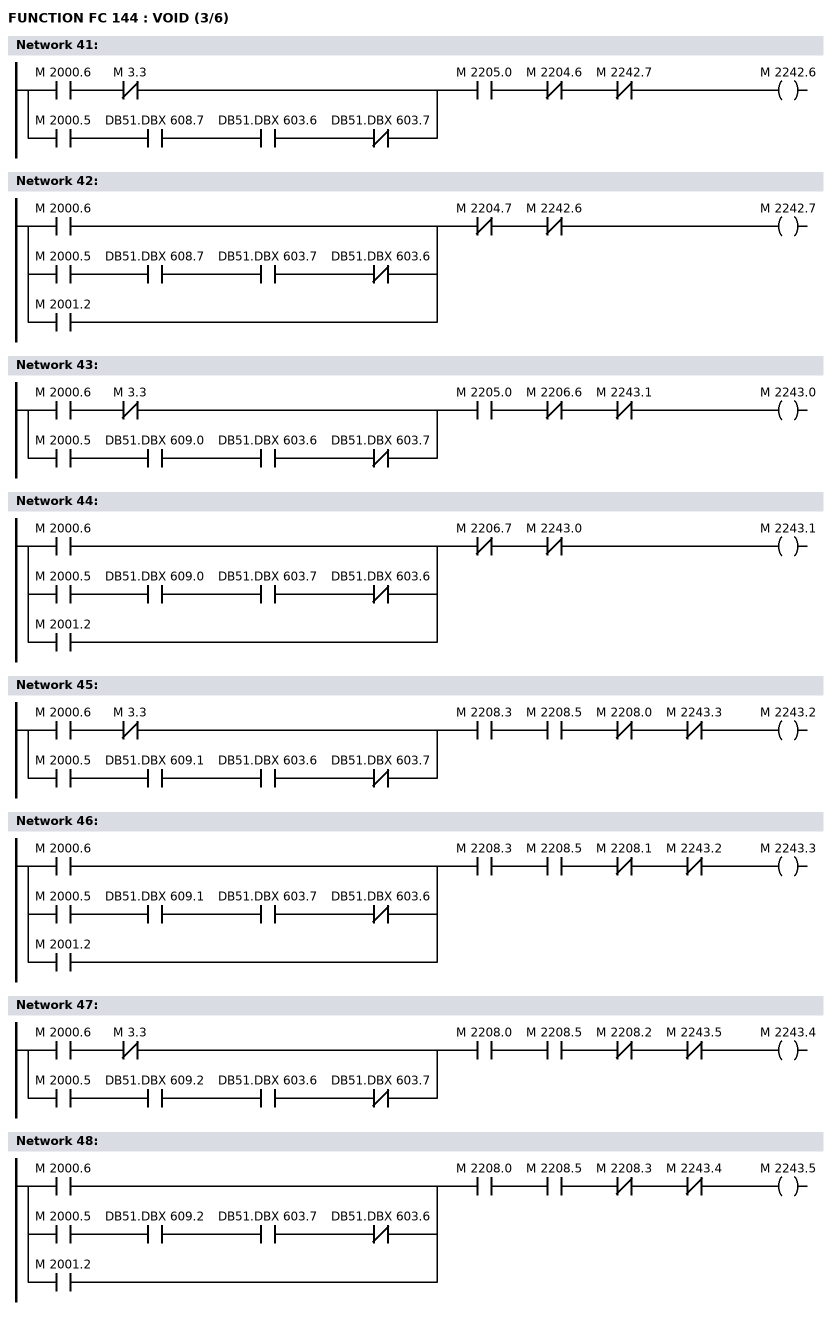

      A(    ;
      A     M   2000.6;
      AN    M      3.3;
      O     ;
      A     M   2000.5;
      A     DB51.DBX  608.7;
      A     DB51.DBX  603.6;
      AN    DB51.DBX  603.7;
      )     ;
      A     M   2205.0;
      AN    M   2204.6;
      AN    M   2242.7;
      =     M   2242.6;
NETWORK
TITLE =

      A(    ;
      O     M   2000.6;
      O     ;
      A     M   2000.5;
      A     DB51.DBX  608.7;
      A     DB51.DBX  603.7;
      AN    DB51.DBX  603.6;
      O     M   2001.2;
      )     ;
      AN    M   2204.7;
      AN    M   2242.6;
      =     M   2242.7;
NETWORK
TITLE =

      A(    ;
      A     M   2000.6;
      AN    M      3.3;
      O     ;
      A     M   2000.5;
      A     DB51.DBX  609.0;
      A     DB51.DBX  603.6;
      AN    DB51.DBX  603.7;
      )     ;
      A     M   2205.0;
      AN    M   2206.6;
      AN    M   2243.1;
      =     M   2243.0;
NETWORK
TITLE =

      A(    ;
      O     M   2000.6;
      O     ;
      A     M   2000.5;
      A     DB51.DBX  609.0;
      A     DB51.DBX  603.7;
      AN    DB51.DBX  603.6;
      O     M   2001.2;
      )     ;
      AN    M   2206.7;
      AN    M   2243.0;
      =     M   2243.1;
NETWORK
TITLE =

      A(    ;
      A     M   2000.6;
      AN    M      3.3;
      O     ;
      A     M   2000.5;
      A     DB51.DBX  609.1;
      A     DB51.DBX  603.6;
      AN    DB51.DBX  603.7;
      )     ;
      A     M   2208.3;
      A     M   2208.5;
      AN    M   2208.0;
      AN    M   2243.3;
      =     M   2243.2;
NETWORK
TITLE =

      A(    ;
      O     M   2000.6;
      O     ;
      A     M   2000.5;
      A     DB51.DBX  609.1;
      A     DB51.DBX  603.7;
      AN    DB51.DBX  603.6;
      O     M   2001.2;
      )     ;
      A     M   2208.3;
      A     M   2208.5;
      AN    M   2208.1;
      AN    M   2243.2;
      =     M   2243.3;
NETWORK
TITLE =

      A(    ;
      A     M   2000.6;
      AN    M      3.3;
      O     ;
      A     M   2000.5;
      A     DB51.DBX  609.2;
      A     DB51.DBX  603.6;
      AN    DB51.DBX  603.7;
      )     ;
      A     M   2208.0;
      A     M   2208.5;
      AN    M   2208.2;
      AN    M   2243.5;
      =     M   2243.4;
NETWORK
TITLE =

      A(    ;
      O     M   2000.6;
      O     ;
      A     M   2000.5;
      A     DB51.DBX  609.2;
      A     DB51.DBX  603.7;
      AN    DB51.DBX  603.6;
      O     M   2001.2;
      )     ;
      A     M   2208.0;
      A     M   2208.5;
      AN    M   2208.3;
      AN    M   2243.4;
      =     M   2243.5;
NETWORK
TITLE =
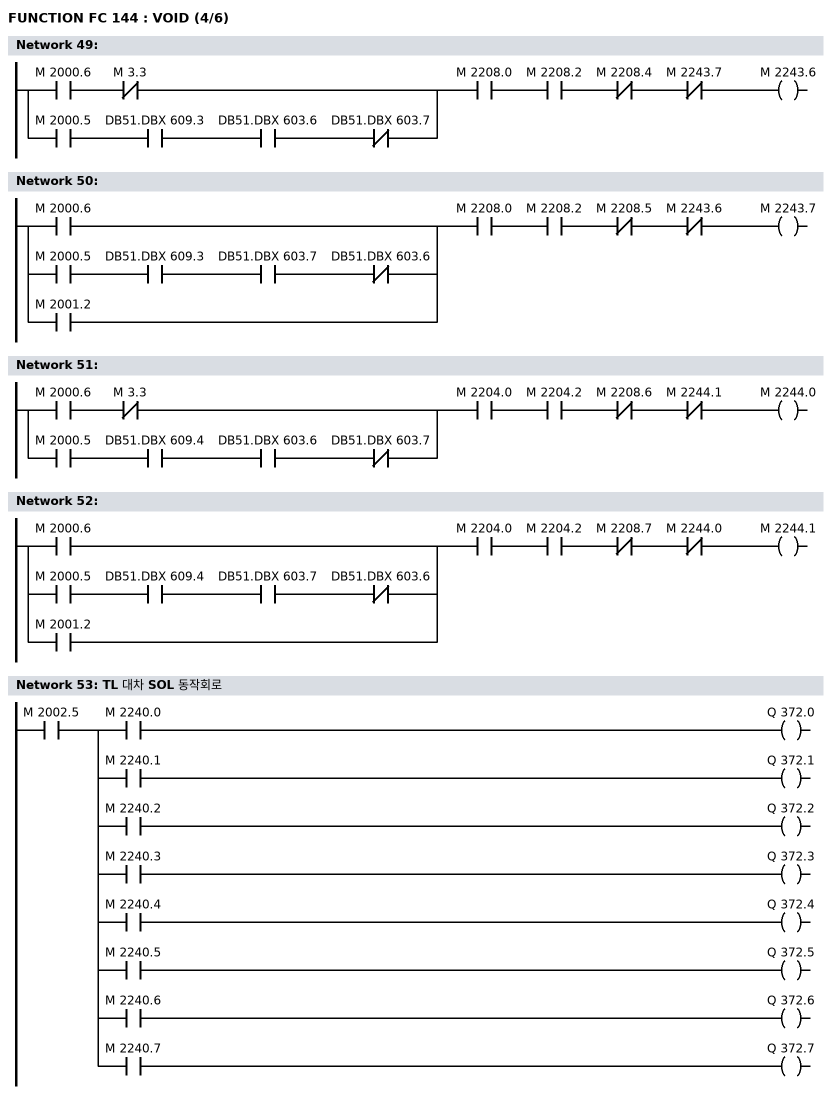

      A(    ;
      A     M   2000.6;
      AN    M      3.3;
      O     ;
      A     M   2000.5;
      A     DB51.DBX  609.3;
      A     DB51.DBX  603.6;
      AN    DB51.DBX  603.7;
      )     ;
      A     M   2208.0;
      A     M   2208.2;
      AN    M   2208.4;
      AN    M   2243.7;
      =     M   2243.6;
NETWORK
TITLE =

      A(    ;
      O     M   2000.6;
      O     ;
      A     M   2000.5;
      A     DB51.DBX  609.3;
      A     DB51.DBX  603.7;
      AN    DB51.DBX  603.6;
      O     M   2001.2;
      )     ;
      A     M   2208.0;
      A     M   2208.2;
      AN    M   2208.5;
      AN    M   2243.6;
      =     M   2243.7;
NETWORK
TITLE =

      A(    ;
      A     M   2000.6;
      AN    M      3.3;
      O     ;
      A     M   2000.5;
      A     DB51.DBX  609.4;
      A     DB51.DBX  603.6;
      AN    DB51.DBX  603.7;
      )     ;
      A     M   2204.0;
      A     M   2204.2;
      AN    M   2208.6;
      AN    M   2244.1;
      =     M   2244.0;
NETWORK
TITLE =

      A(    ;
      O     M   2000.6;
      O     ;
      A     M   2000.5;
      A     DB51.DBX  609.4;
      A     DB51.DBX  603.7;
      AN    DB51.DBX  603.6;
      O     M   2001.2;
      )     ;
      A     M   2204.0;
      A     M   2204.2;
      AN    M   2208.7;
      AN    M   2244.0;
      =     M   2244.1;
NETWORK
TITLE =TL 대차 SOL 동작회로

      A     M   2002.5;
      =     L      0.0;
      A     L      0.0;
      A     M   2240.0;
      =     Q    372.0;
      A     L      0.0;
      A     M   2240.1;
      =     Q    372.1;
      A     L      0.0;
      A     M   2240.2;
      =     Q    372.2;
      A     L      0.0;
      A     M   2240.3;
      =     Q    372.3;
      A     L      0.0;
      A     M   2240.4;
      =     Q    372.4;
      A     L      0.0;
      A     M   2240.5;
      =     Q    372.5;
      A     L      0.0;
      A     M   2240.6;
      =     Q    372.6;
      A     L      0.0;
      A     M   2240.7;
      =     Q    372.7;
NETWORK
TITLE =
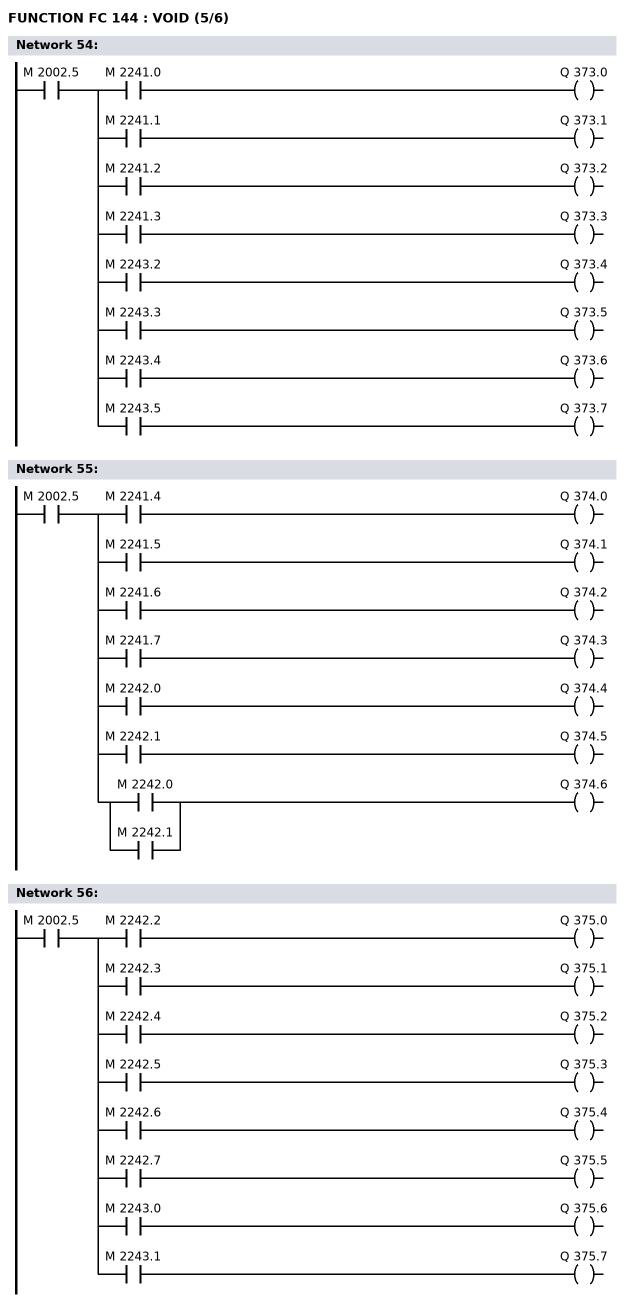

      A     M   2002.5;
      =     L      0.0;
      A     L      0.0;
      A     M   2241.0;
      =     Q    373.0;
      A     L      0.0;
      A     M   2241.1;
      =     Q    373.1;
      A     L      0.0;
      A     M   2241.2;
      =     Q    373.2;
      A     L      0.0;
      A     M   2241.3;
      =     Q    373.3;
      A     L      0.0;
      A     M   2243.2;
      =     Q    373.4;
      A     L      0.0;
      A     M   2243.3;
      =     Q    373.5;
      A     L      0.0;
      A     M   2243.4;
      =     Q    373.6;
      A     L      0.0;
      A     M   2243.5;
      =     Q    373.7;
NETWORK
TITLE =

      A     M   2002.5;
      =     L      0.0;
      A     L      0.0;
      A     M   2241.4;
      =     Q    374.0;
      A     L      0.0;
      A     M   2241.5;
      =     Q    374.1;
      A     L      0.0;
      A     M   2241.6;
      =     Q    374.2;
      A     L      0.0;
      A     M   2241.7;
      =     Q    374.3;
      A     L      0.0;
      A     M   2242.0;
      =     Q    374.4;
      A     L      0.0;
      A     M   2242.1;
      =     Q    374.5;
      A     L      0.0;
      A(    ;
      O     M   2242.0;
      O     M   2242.1;
      )     ;
      =     Q    374.6;
NETWORK
TITLE =

      A     M   2002.5;
      =     L      0.0;
      A     L      0.0;
      A     M   2242.2;
      =     Q    375.0;
      A     L      0.0;
      A     M   2242.3;
      =     Q    375.1;
      A     L      0.0;
      A     M   2242.4;
      =     Q    375.2;
      A     L      0.0;
      A     M   2242.5;
      =     Q    375.3;
      A     L      0.0;
      A     M   2242.6;
      =     Q    375.4;
      A     L      0.0;
      A     M   2242.7;
      =     Q    375.5;
      A     L      0.0;
      A     M   2243.0;
      =     Q    375.6;
      A     L      0.0;
      A     M   2243.1;
      =     Q    375.7;
NETWORK
TITLE =
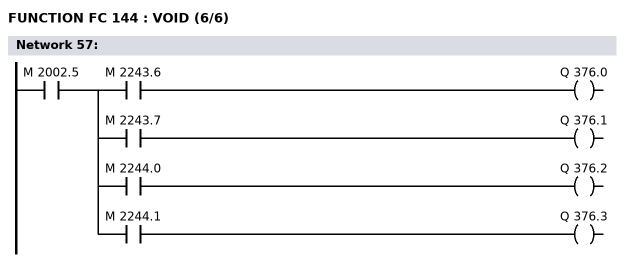

      A     M   2002.5;
      =     L      0.0;
      A     L      0.0;
      A     M   2243.6;
      =     Q    376.0;
      A     L      0.0;
      A     M   2243.7;
      =     Q    376.1;
      A     L      0.0;
      A     M   2244.0;
      =     Q    376.2;
      A     L      0.0;
      A     M   2244.1;
      =     Q    376.3;
END_FUNCTION

FUNCTION FC 145 : VOID
TITLE =
VERSION : 0.1

BEGIN
NETWORK
TITLE =
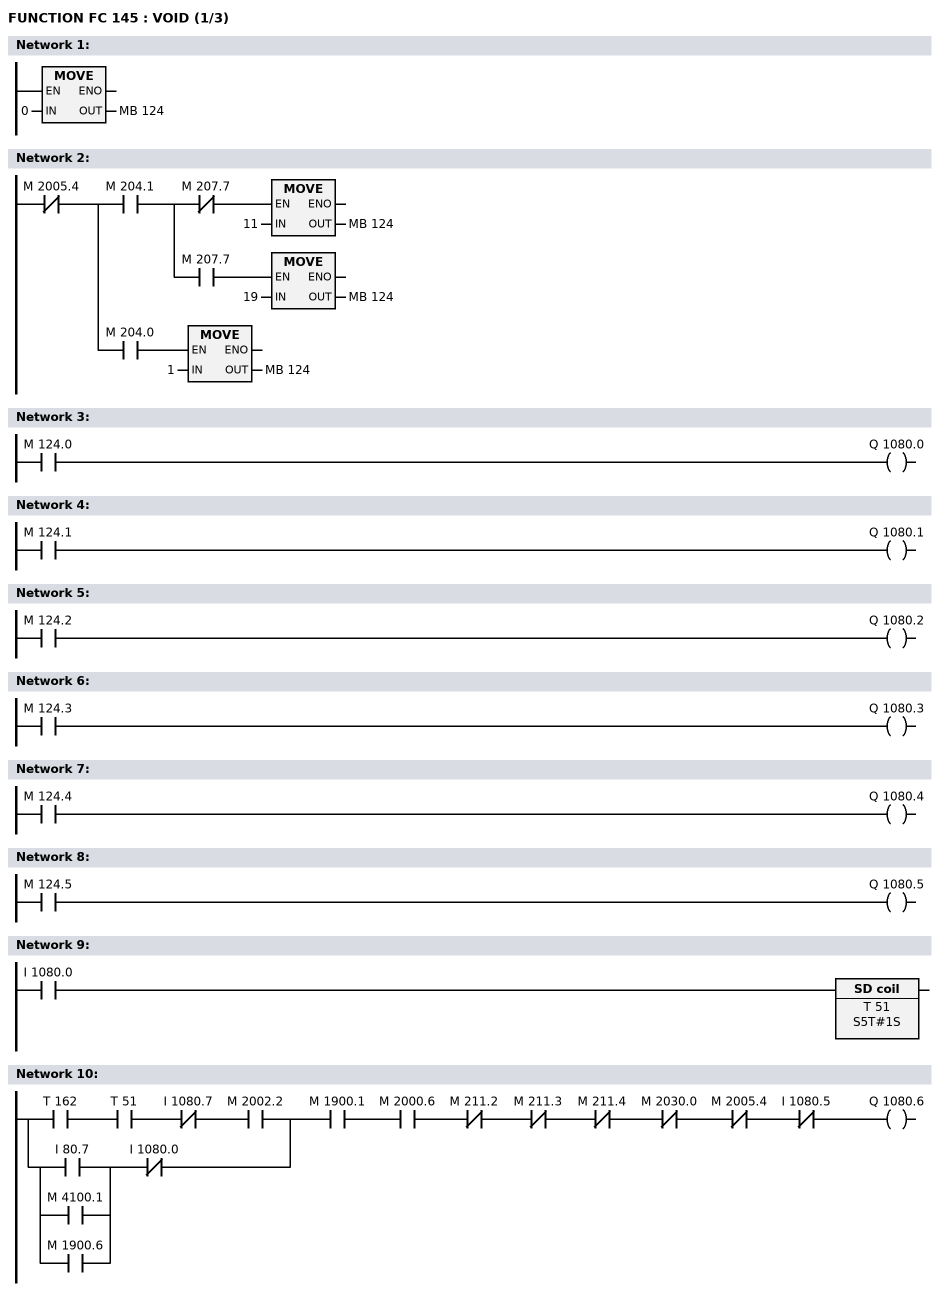

      L     0;
      T     MB   124;
      NOP   0;
NETWORK
TITLE =

      AN    M   2005.4;
      =     L      0.0;
      A     L      0.0;
      A     M    204.1;
      =     L      0.1;
      A     L      0.1;
      AN    M    207.7;
      JNB   _001;
      L     11;
      T     MB   124;
_001: NOP   0;
      A     L      0.1;
      A     M    207.7;
      JNB   _002;
      L     19;
      T     MB   124;
_002: NOP   0;
      A     L      0.0;
      A     M    204.0;
      JNB   _003;
      L     1;
      T     MB   124;
_003: NOP   0;
NETWORK
TITLE =

      A     M    124.0;
      =     Q   1080.0;
NETWORK
TITLE =

      A     M    124.1;
      =     Q   1080.1;
NETWORK
TITLE =

      A     M    124.2;
      =     Q   1080.2;
NETWORK
TITLE =

      A     M    124.3;
      =     Q   1080.3;
NETWORK
TITLE =

      A     M    124.4;
      =     Q   1080.4;
NETWORK
TITLE =

      A     M    124.5;
      =     Q   1080.5;
NETWORK
TITLE =

      A     I   1080.0;
      L     S5T#1S;
      SD    T     51;
NETWORK
TITLE =

      A(    ;
      A     T    162;
      A     T     51;
      AN    I   1080.7;
      A     M   2002.2;
      O     ;
      A(    ;
      O     I     80.7;
      O     M   4100.1;
      O     M   1900.6;
      )     ;
      AN    I   1080.0;
      )     ;
      A     M   1900.1;
      A     M   2000.6;
      AN    M    211.2;
      AN    M    211.3;
      AN    M    211.4;
      AN    M   2030.0;
      AN    M   2005.4;
      AN    I   1080.5;
      =     Q   1080.6;
NETWORK
TITLE =
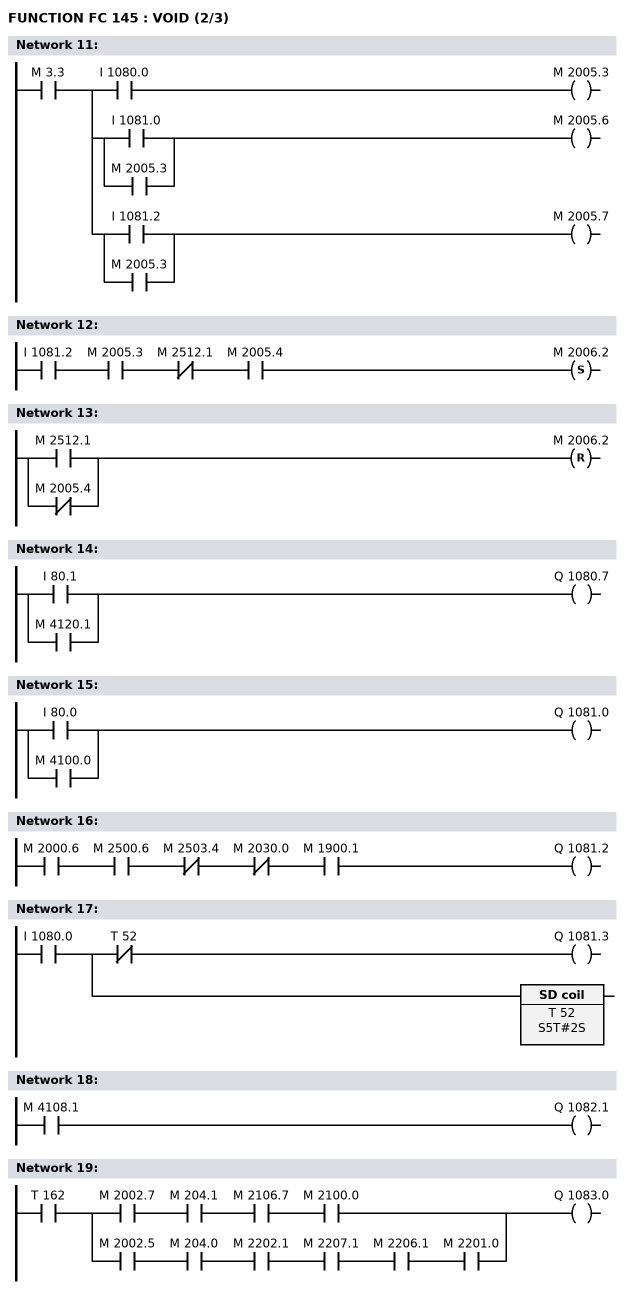

      A     M      3.3;
      =     L      0.0;
      A     L      0.0;
      A     I   1080.0;
      =     M   2005.3;
      A     L      0.0;
      A(    ;
      O     I   1081.0;
      O     M   2005.3;
      )     ;
      =     M   2005.6;
      A     L      0.0;
      A(    ;
      O     I   1081.2;
      O     M   2005.3;
      )     ;
      =     M   2005.7;
NETWORK
TITLE =

      A     I   1081.2;
      A     M   2005.3;
      AN    M   2512.1;
      A     M   2005.4;
      S     M   2006.2;
NETWORK
TITLE =

      O     M   2512.1;
      ON    M   2005.4;
      R     M   2006.2;
NETWORK
TITLE =

      O     I     80.1;
      O     M   4120.1;
      =     Q   1080.7;
NETWORK
TITLE =

      O     I     80.0;
      O     M   4100.0;
      =     Q   1081.0;
NETWORK
TITLE =

      A     M   2000.6;
      A     M   2500.6;
      AN    M   2503.4;
      AN    M   2030.0;
      A     M   1900.1;
      =     Q   1081.2;
NETWORK
TITLE =

      A     I   1080.0;
      =     L      0.0;
      A     L      0.0;
      AN    T     52;
      =     Q   1081.3;
      A     L      0.0;
      BLD   102;
      L     S5T#2S;
      SD    T     52;
NETWORK
TITLE =

      A     M   4108.1;
      =     Q   1082.1;
NETWORK
TITLE =

      A     T    162;
      A(    ;
      A     M   2002.7;
      A     M    204.1;
      A     M   2106.7;
      A     M   2100.0;
      O     ;
      A     M   2002.5;
      A     M    204.0;
      A     M   2202.1;
      A     M   2207.1;
      A     M   2206.1;
      A     M   2201.0;
      )     ;
      =     Q   1083.0;
NETWORK
TITLE =
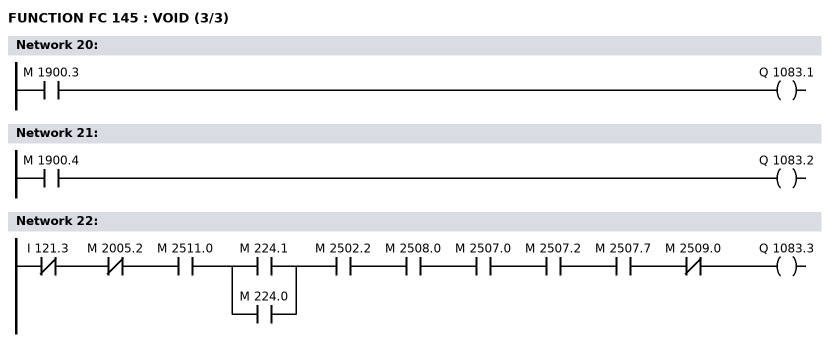

      A     M   1900.3;
      =     Q   1083.1;
NETWORK
TITLE =

      A     M   1900.4;
      =     Q   1083.2;
NETWORK
TITLE =

      AN    I    121.3;
      AN    M   2005.2;
      A     M   2511.0;
      A(    ;
      O     M    224.1;
      O     M    224.0;
      )     ;
      A     M   2502.2;
      A     M   2508.0;
      A     M   2507.0;
      A     M   2507.2;
      A     M   2507.7;
      AN    M   2509.0;
      =     Q   1083.3;
END_FUNCTION

FUNCTION_BLOCK FB 150
TITLE =
VERSION : 0.1


VAR
  S_UP_DL_MODE : FB 402;
END_VAR
BEGIN
NETWORK
TITLE =
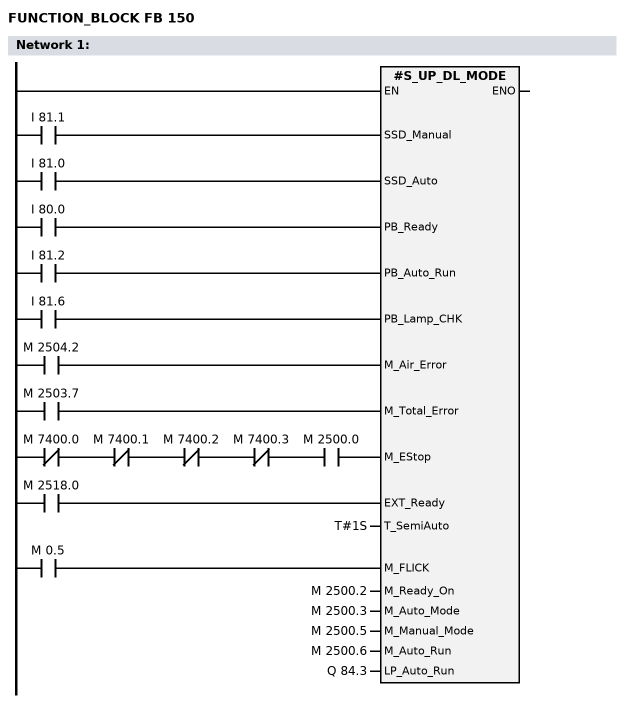

      A     I     81.1;
      =     L      0.0;
      BLD   103;
      A     I     81.0;
      =     L      0.1;
      BLD   103;
      A     I     80.0;
      =     L      0.2;
      BLD   103;
      A     I     81.2;
      =     L      0.3;
      BLD   103;
      A     I     81.6;
      =     L      0.6;
      BLD   103;
      A     M   2504.2;
      =     L      0.7;
      BLD   103;
      A     M   2503.7;
      =     L      1.1;
      BLD   103;
      AN    M   7400.0;
      AN    M   7400.1;
      AN    M   7400.2;
      AN    M   7400.3;
      A     M   2500.0;
      =     L      1.2;
      BLD   103;
      A     M   2518.0;
      =     L      1.3;
      BLD   103;
      A     M      0.5;
      =     L      1.5;
      BLD   103;
      CALL #S_UP_DL_MODE (
           SSD_Manual               := L      0.0,
           SSD_Auto                 := L      0.1,
           PB_Ready                 := L      0.2,
           PB_Auto_Run              := L      0.3,
           PB_Lamp_CHK              := L      0.6,
           M_Air_Error              := L      0.7,
           M_Total_Error            := L      1.1,
           M_EStop                  := L      1.2,
           EXT_Ready                := L      1.3,
           T_SemiAuto               := T#1S,
           M_FLICK                  := L      1.5,
           M_Ready_On               := M   2500.2,
           M_Auto_Mode              := M   2500.3,
           M_Manual_Mode            := M   2500.5,
           M_Auto_Run               := M   2500.6,
           LP_Auto_Run              := Q     84.3);
      NOP   0;
END_FUNCTION_BLOCK

DATA_BLOCK DB 150
TITLE =
VERSION : 0.0

 FB 150
BEGIN
   S_UP_DL_MODE.SSD_Manual := FALSE;
   S_UP_DL_MODE.SSD_Auto := TRUE;
   S_UP_DL_MODE.PB_Ready := FALSE;
   S_UP_DL_MODE.PB_Auto_Run := FALSE;
   S_UP_DL_MODE.PB_Remote_Ready := FALSE;
   S_UP_DL_MODE.PB_Remote_Auto_Run := FALSE;
   S_UP_DL_MODE.PB_Lamp_CHK := FALSE;
   S_UP_DL_MODE.M_Air_Error := FALSE;
   S_UP_DL_MODE.M_Water_Error := FALSE;
   S_UP_DL_MODE.M_Total_Error := FALSE;
   S_UP_DL_MODE.M_EStop := TRUE;
   S_UP_DL_MODE.EXT_Ready := TRUE;
   S_UP_DL_MODE.EXT_Auto := FALSE;
   S_UP_DL_MODE.T_SemiAuto := T#1S;
   S_UP_DL_MODE.M_FLICK := FALSE;
   S_UP_DL_MODE.M_Ready_On := TRUE;
   S_UP_DL_MODE.M_Auto_Mode := TRUE;
   S_UP_DL_MODE.M_SemiAuto_Mode := FALSE;
   S_UP_DL_MODE.M_Manual_Mode := FALSE;
   S_UP_DL_MODE.M_Auto_Run := TRUE;
   S_UP_DL_MODE.LP_Ready_On := TRUE;
   S_UP_DL_MODE.LP_Auto_Run := TRUE;
   S_UP_DL_MODE.AUTO_MODE_DELAY.IN := FALSE;
   S_UP_DL_MODE.AUTO_MODE_DELAY.PT := T#0MS;
   S_UP_DL_MODE.AUTO_MODE_DELAY.Q := FALSE;
   S_UP_DL_MODE.AUTO_MODE_DELAY.ET := T#0MS;
   S_UP_DL_MODE.AUTO_MODE_DELAY.STATE := B#16#0;
   S_UP_DL_MODE.AUTO_MODE_DELAY.STIME := T#0MS;
   S_UP_DL_MODE.AUTO_MODE_DELAY.ATIME := T#0MS;
   S_UP_DL_MODE.SEMI_AUTO_DELAY.IN := FALSE;
   S_UP_DL_MODE.SEMI_AUTO_DELAY.PT := T#1S;
   S_UP_DL_MODE.SEMI_AUTO_DELAY.Q := FALSE;
   S_UP_DL_MODE.SEMI_AUTO_DELAY.ET := T#0MS;
   S_UP_DL_MODE.SEMI_AUTO_DELAY.STATE := B#16#0;
   S_UP_DL_MODE.SEMI_AUTO_DELAY.STIME := T#22D16H36M7S51MS;
   S_UP_DL_MODE.SEMI_AUTO_DELAY.ATIME := T#22D16H36M7S75MS;
   S_UP_DL_MODE.MANUAL_DELAY.IN := FALSE;
   S_UP_DL_MODE.MANUAL_DELAY.PT := T#0MS;
   S_UP_DL_MODE.MANUAL_DELAY.Q := FALSE;
   S_UP_DL_MODE.MANUAL_DELAY.ET := T#0MS;
   S_UP_DL_MODE.MANUAL_DELAY.STATE := B#16#0;
   S_UP_DL_MODE.MANUAL_DELAY.STIME := T#0MS;
   S_UP_DL_MODE.MANUAL_DELAY.ATIME := T#0MS;
END_DATA_BLOCK

FUNCTION FC 150 : VOID
TITLE =
VERSION : 0.1

BEGIN
NETWORK
TITLE =
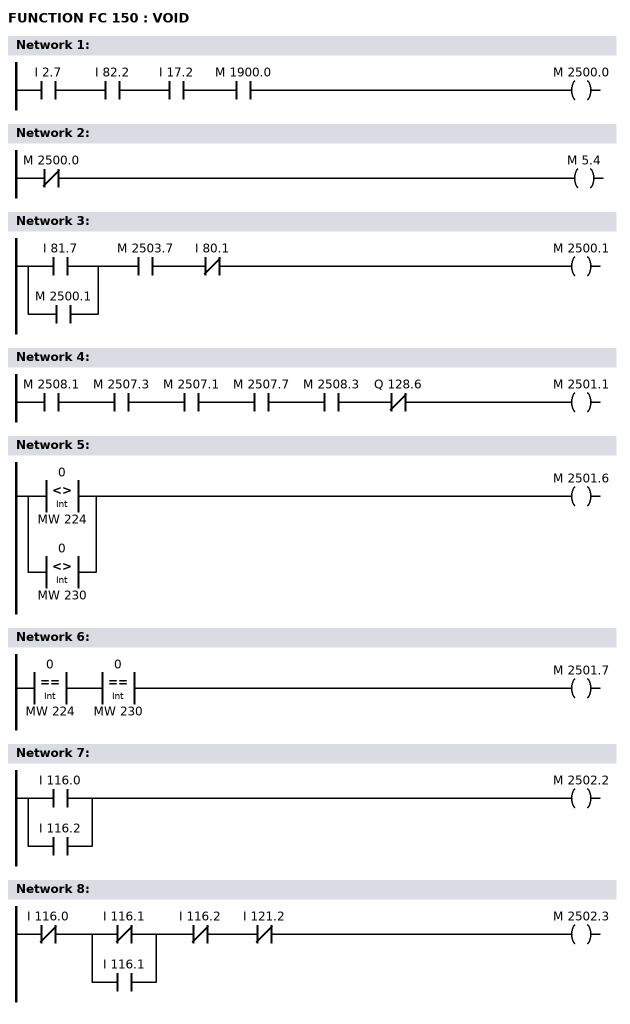

      A     I      2.7;
      A     I     82.2;
      A     I     17.2;
      A     M   1900.0;
      =     M   2500.0;
NETWORK
TITLE =

      AN    M   2500.0;
      =     M      5.4;
NETWORK
TITLE =

      A(    ;
      O     I     81.7;
      O     M   2500.1;
      )     ;
      A     M   2503.7;
      AN    I     80.1;
      =     M   2500.1;
NETWORK
TITLE =

      A     M   2508.1;
      A     M   2507.3;
      A     M   2507.1;
      A     M   2507.7;
      A     M   2508.3;
      AN    Q    128.6;
      =     M   2501.1;
NETWORK
TITLE =

      O(    ;
      L     0;
      L     MW   224;
      <>I   ;
      )     ;
      O(    ;
      L     0;
      L     MW   230;
      <>I   ;
      )     ;
      =     M   2501.6;
NETWORK
TITLE =

      A(    ;
      L     0;
      L     MW   224;
      ==I   ;
      )     ;
      A(    ;
      L     0;
      L     MW   230;
      ==I   ;
      )     ;
      =     M   2501.7;
NETWORK
TITLE =

      O     I    116.0;
      O     I    116.2;
      =     M   2502.2;
NETWORK
TITLE =

      AN    I    116.0;
      A(    ;
      ON    I    116.1;
      O     I    116.1;
      )     ;
      AN    I    116.2;
      AN    I    121.2;
      =     M   2502.3;
END_FUNCTION

FUNCTION_BLOCK FB 151
TITLE =
VERSION : 0.1


VAR
  UP_DL_DAECHA_CLAMP : FB 424;
  UP_DL_AIR_ELE_UP_DOWN : FB 424;
  UP_DL_AIR_ELE_ADV_RET : FB 424;
  UP_DL_LIFT_LOCK : FB 424;
  UP_DL_LIFT : FB 424;
END_VAR
BEGIN
NETWORK
TITLE =
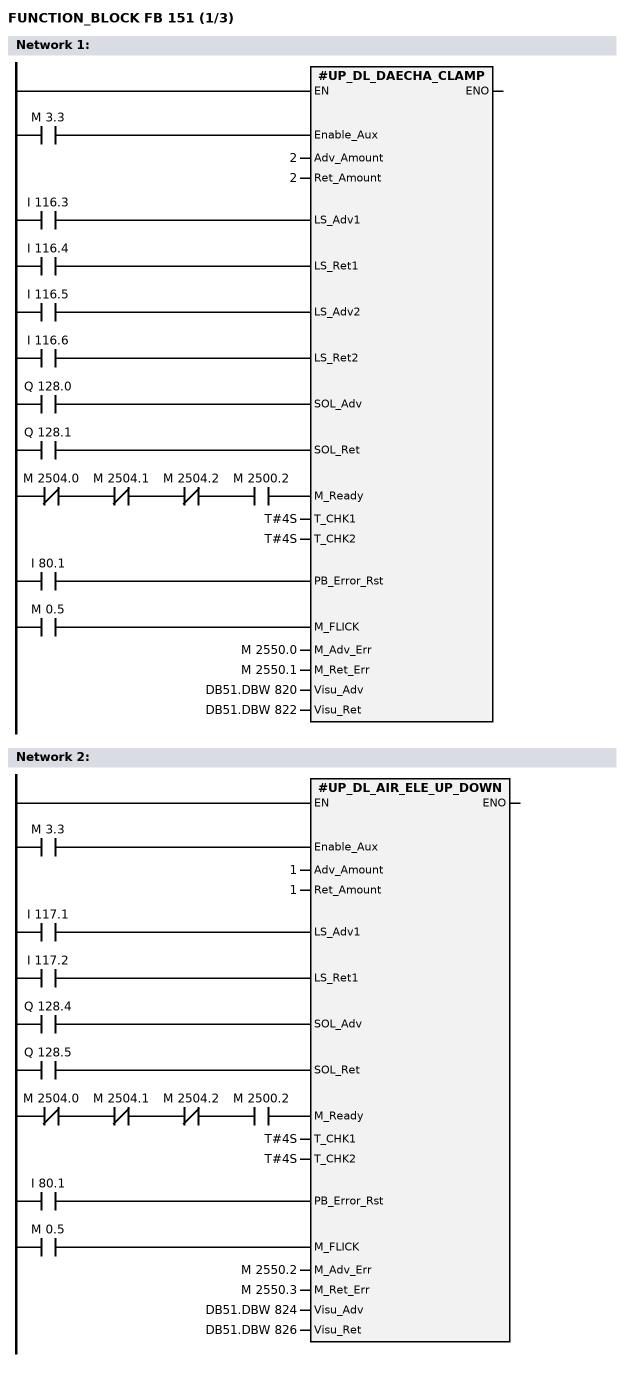

      A     M      3.3;
      =     L      0.0;
      BLD   103;
      A     I    116.3;
      =     L      0.1;
      BLD   103;
      A     I    116.4;
      =     L      0.2;
      BLD   103;
      A     I    116.5;
      =     L      0.3;
      BLD   103;
      A     I    116.6;
      =     L      0.4;
      BLD   103;
      A     Q    128.0;
      =     L      1.1;
      BLD   103;
      A     Q    128.1;
      =     L      1.2;
      BLD   103;
      AN    M   2504.0;
      AN    M   2504.1;
      AN    M   2504.2;
      A     M   2500.2;
      =     L      1.3;
      BLD   103;
      A     I     80.1;
      =     L      1.5;
      BLD   103;
      A     M      0.5;
      =     L      1.6;
      BLD   103;
      CALL #UP_DL_DAECHA_CLAMP (
           Enable_Aux               := L      0.0,
           Adv_Amount               := 2,
           Ret_Amount               := 2,
           LS_Adv1                  := L      0.1,
           LS_Ret1                  := L      0.2,
           LS_Adv2                  := L      0.3,
           LS_Ret2                  := L      0.4,
           SOL_Adv                  := L      1.1,
           SOL_Ret                  := L      1.2,
           M_Ready                  := L      1.3,
           T_CHK1                   := T#4S,
           T_CHK2                   := T#4S,
           PB_Error_Rst             := L      1.5,
           M_FLICK                  := L      1.6,
           M_Adv_Err                := M   2550.0,
           M_Ret_Err                := M   2550.1,
           Visu_Adv                 := DB51.DBW  820,
           Visu_Ret                 := DB51.DBW  822);
      NOP   0;
NETWORK
TITLE =

      A     M      3.3;
      =     L      0.0;
      BLD   103;
      A     I    117.1;
      =     L      0.1;
      BLD   103;
      A     I    117.2;
      =     L      0.2;
      BLD   103;
      A     Q    128.4;
      =     L      1.1;
      BLD   103;
      A     Q    128.5;
      =     L      1.2;
      BLD   103;
      AN    M   2504.0;
      AN    M   2504.1;
      AN    M   2504.2;
      A     M   2500.2;
      =     L      1.3;
      BLD   103;
      A     I     80.1;
      =     L      1.5;
      BLD   103;
      A     M      0.5;
      =     L      1.6;
      BLD   103;
      CALL #UP_DL_AIR_ELE_UP_DOWN (
           Enable_Aux               := L      0.0,
           Adv_Amount               := 1,
           Ret_Amount               := 1,
           LS_Adv1                  := L      0.1,
           LS_Ret1                  := L      0.2,
           SOL_Adv                  := L      1.1,
           SOL_Ret                  := L      1.2,
           M_Ready                  := L      1.3,
           T_CHK1                   := T#4S,
           T_CHK2                   := T#4S,
           PB_Error_Rst             := L      1.5,
           M_FLICK                  := L      1.6,
           M_Adv_Err                := M   2550.2,
           M_Ret_Err                := M   2550.3,
           Visu_Adv                 := DB51.DBW  824,
           Visu_Ret                 := DB51.DBW  826);
      NOP   0;
NETWORK
TITLE =
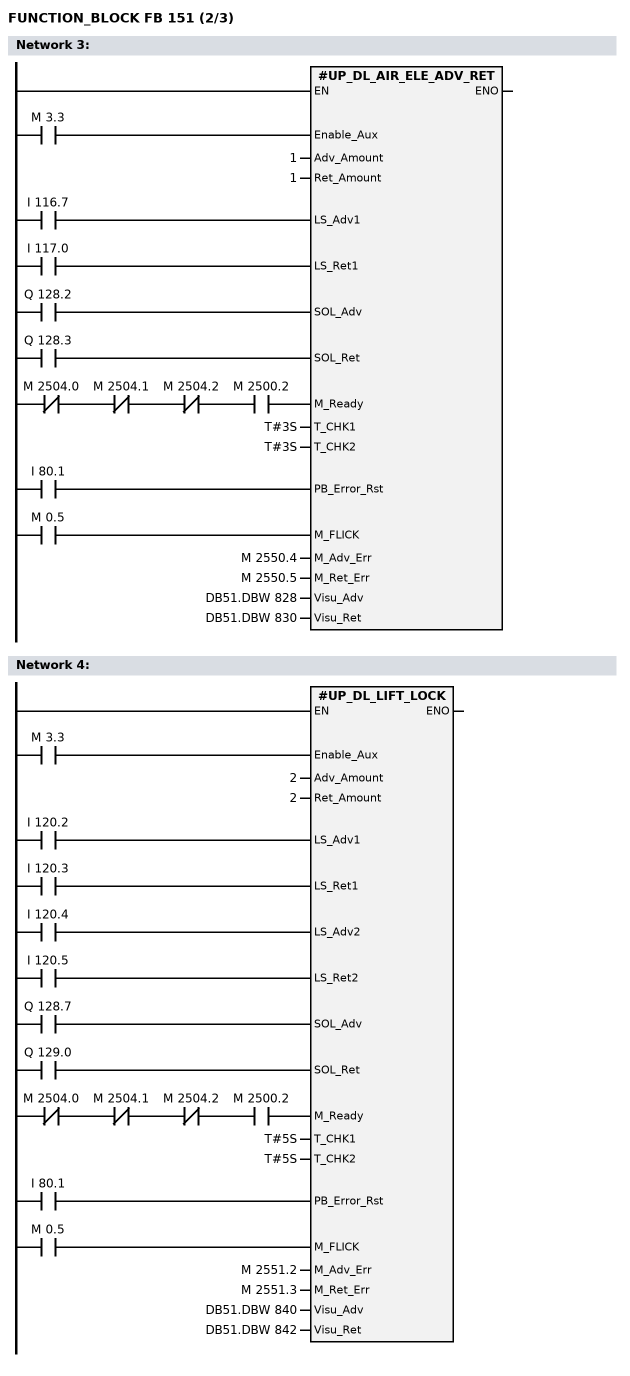

      A     M      3.3;
      =     L      0.0;
      BLD   103;
      A     I    116.7;
      =     L      0.1;
      BLD   103;
      A     I    117.0;
      =     L      0.2;
      BLD   103;
      A     Q    128.2;
      =     L      1.1;
      BLD   103;
      A     Q    128.3;
      =     L      1.2;
      BLD   103;
      AN    M   2504.0;
      AN    M   2504.1;
      AN    M   2504.2;
      A     M   2500.2;
      =     L      1.3;
      BLD   103;
      A     I     80.1;
      =     L      1.5;
      BLD   103;
      A     M      0.5;
      =     L      1.6;
      BLD   103;
      CALL #UP_DL_AIR_ELE_ADV_RET (
           Enable_Aux               := L      0.0,
           Adv_Amount               := 1,
           Ret_Amount               := 1,
           LS_Adv1                  := L      0.1,
           LS_Ret1                  := L      0.2,
           SOL_Adv                  := L      1.1,
           SOL_Ret                  := L      1.2,
           M_Ready                  := L      1.3,
           T_CHK1                   := T#3S,
           T_CHK2                   := T#3S,
           PB_Error_Rst             := L      1.5,
           M_FLICK                  := L      1.6,
           M_Adv_Err                := M   2550.4,
           M_Ret_Err                := M   2550.5,
           Visu_Adv                 := DB51.DBW  828,
           Visu_Ret                 := DB51.DBW  830);
      NOP   0;
NETWORK
TITLE =

      A     M      3.3;
      =     L      0.0;
      BLD   103;
      A     I    120.2;
      =     L      0.1;
      BLD   103;
      A     I    120.3;
      =     L      0.2;
      BLD   103;
      A     I    120.4;
      =     L      0.3;
      BLD   103;
      A     I    120.5;
      =     L      0.4;
      BLD   103;
      A     Q    128.7;
      =     L      1.1;
      BLD   103;
      A     Q    129.0;
      =     L      1.2;
      BLD   103;
      AN    M   2504.0;
      AN    M   2504.1;
      AN    M   2504.2;
      A     M   2500.2;
      =     L      1.3;
      BLD   103;
      A     I     80.1;
      =     L      1.5;
      BLD   103;
      A     M      0.5;
      =     L      1.6;
      BLD   103;
      CALL #UP_DL_LIFT_LOCK (
           Enable_Aux               := L      0.0,
           Adv_Amount               := 2,
           Ret_Amount               := 2,
           LS_Adv1                  := L      0.1,
           LS_Ret1                  := L      0.2,
           LS_Adv2                  := L      0.3,
           LS_Ret2                  := L      0.4,
           SOL_Adv                  := L      1.1,
           SOL_Ret                  := L      1.2,
           M_Ready                  := L      1.3,
           T_CHK1                   := T#5S,
           T_CHK2                   := T#5S,
           PB_Error_Rst             := L      1.5,
           M_FLICK                  := L      1.6,
           M_Adv_Err                := M   2551.2,
           M_Ret_Err                := M   2551.3,
           Visu_Adv                 := DB51.DBW  840,
           Visu_Ret                 := DB51.DBW  842);
      NOP   0;
NETWORK
TITLE =
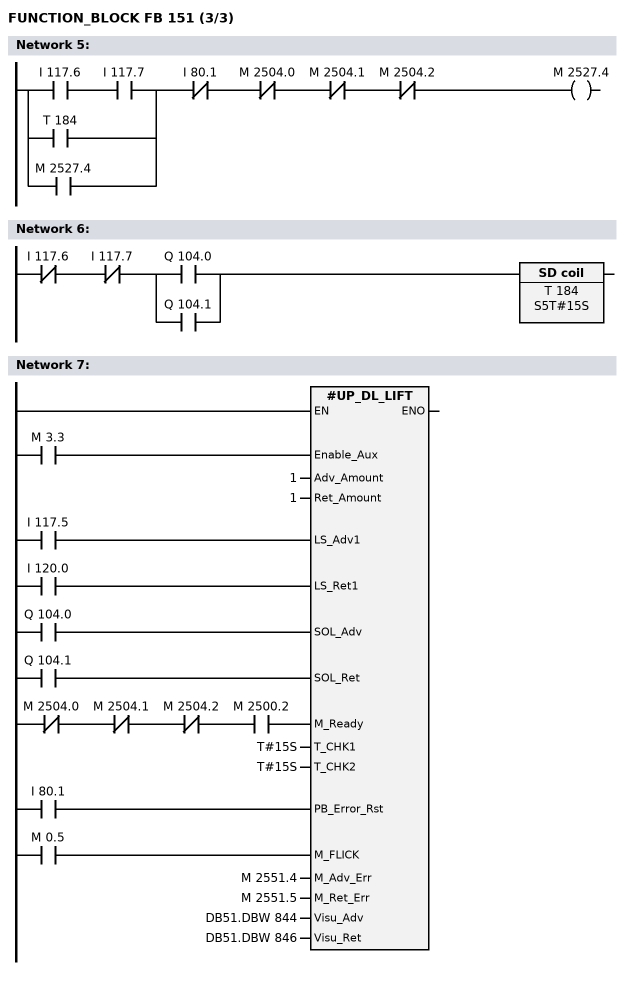

      A(    ;
      A     I    117.6;
      A     I    117.7;
      O     T    184;
      O     M   2527.4;
      )     ;
      AN    I     80.1;
      AN    M   2504.0;
      AN    M   2504.1;
      AN    M   2504.2;
      =     M   2527.4;
NETWORK
TITLE =

      AN    I    117.6;
      AN    I    117.7;
      A(    ;
      O     Q    104.0;
      O     Q    104.1;
      )     ;
      L     S5T#15S;
      SD    T    184;
NETWORK
TITLE =

      A     M      3.3;
      =     L      0.0;
      BLD   103;
      A     I    117.5;
      =     L      0.1;
      BLD   103;
      A     I    120.0;
      =     L      0.2;
      BLD   103;
      A     Q    104.0;
      =     L      1.1;
      BLD   103;
      A     Q    104.1;
      =     L      1.2;
      BLD   103;
      AN    M   2504.0;
      AN    M   2504.1;
      AN    M   2504.2;
      A     M   2500.2;
      =     L      1.3;
      BLD   103;
      A     I     80.1;
      =     L      1.5;
      BLD   103;
      A     M      0.5;
      =     L      1.6;
      BLD   103;
      CALL #UP_DL_LIFT (
           Enable_Aux               := L      0.0,
           Adv_Amount               := 1,
           Ret_Amount               := 1,
           LS_Adv1                  := L      0.1,
           LS_Ret1                  := L      0.2,
           SOL_Adv                  := L      1.1,
           SOL_Ret                  := L      1.2,
           M_Ready                  := L      1.3,
           T_CHK1                   := T#15S,
           T_CHK2                   := T#15S,
           PB_Error_Rst             := L      1.5,
           M_FLICK                  := L      1.6,
           M_Adv_Err                := M   2551.4,
           M_Ret_Err                := M   2551.5,
           Visu_Adv                 := DB51.DBW  844,
           Visu_Ret                 := DB51.DBW  846);
      NOP   0;
END_FUNCTION_BLOCK

DATA_BLOCK DB 151
TITLE =
VERSION : 0.0

 FB 151
BEGIN
   UP_DL_DAECHA_CLAMP.Enable_Aux := TRUE;
   UP_DL_DAECHA_CLAMP.Adv_Amount := 2;
   UP_DL_DAECHA_CLAMP.Ret_Amount := 2;
   UP_DL_DAECHA_CLAMP.LS_Adv1 := FALSE;
   UP_DL_DAECHA_CLAMP.LS_Ret1 := TRUE;
   UP_DL_DAECHA_CLAMP.LS_Adv2 := FALSE;
   UP_DL_DAECHA_CLAMP.LS_Ret2 := TRUE;
   UP_DL_DAECHA_CLAMP.LS_Adv3 := FALSE;
   UP_DL_DAECHA_CLAMP.LS_Ret3 := FALSE;
   UP_DL_DAECHA_CLAMP.LS_Adv4 := FALSE;
   UP_DL_DAECHA_CLAMP.LS_Ret4 := FALSE;
   UP_DL_DAECHA_CLAMP.SOL_Adv := FALSE;
   UP_DL_DAECHA_CLAMP.SOL_Ret := FALSE;
   UP_DL_DAECHA_CLAMP.M_Ready := TRUE;
   UP_DL_DAECHA_CLAMP.T_CHK1 := T#4S;
   UP_DL_DAECHA_CLAMP.T_CHK2 := T#4S;
   UP_DL_DAECHA_CLAMP.PB_Lamp_CHK := FALSE;
   UP_DL_DAECHA_CLAMP.PB_Error_Rst := FALSE;
   UP_DL_DAECHA_CLAMP.M_FLICK := TRUE;
   UP_DL_DAECHA_CLAMP.M_Adv_Err := FALSE;
   UP_DL_DAECHA_CLAMP.M_Ret_Err := FALSE;
   UP_DL_DAECHA_CLAMP.LP_Adv := FALSE;
   UP_DL_DAECHA_CLAMP.LP_Ret := TRUE;
   UP_DL_DAECHA_CLAMP.Visu_Adv := W#16#0;
   UP_DL_DAECHA_CLAMP.Visu_Ret := W#16#700;
   UP_DL_DAECHA_CLAMP.Error_T1.IN := FALSE;
   UP_DL_DAECHA_CLAMP.Error_T1.PT := T#4S;
   UP_DL_DAECHA_CLAMP.Error_T1.Q := FALSE;
   UP_DL_DAECHA_CLAMP.Error_T1.ET := T#0MS;
   UP_DL_DAECHA_CLAMP.Error_T1.STATE := B#16#0;
   UP_DL_DAECHA_CLAMP.Error_T1.STIME := T#23D5H8M58S224MS;
   UP_DL_DAECHA_CLAMP.Error_T1.ATIME := T#23D5H8M59S528MS;
   UP_DL_DAECHA_CLAMP.Error_T2.IN := FALSE;
   UP_DL_DAECHA_CLAMP.Error_T2.PT := T#4S;
   UP_DL_DAECHA_CLAMP.Error_T2.Q := FALSE;
   UP_DL_DAECHA_CLAMP.Error_T2.ET := T#0MS;
   UP_DL_DAECHA_CLAMP.Error_T2.STATE := B#16#0;
   UP_DL_DAECHA_CLAMP.Error_T2.STIME := T#0MS;
   UP_DL_DAECHA_CLAMP.Error_T2.ATIME := T#0MS;
   UP_DL_DAECHA_CLAMP.CHK_Aux1 := FALSE;
   UP_DL_DAECHA_CLAMP.CHK_Aux2 := FALSE;
   UP_DL_DAECHA_CLAMP.Error_T1_DN := FALSE;
   UP_DL_DAECHA_CLAMP.Error_T2_DN := FALSE;
   UP_DL_DAECHA_CLAMP.Adv_Memo := FALSE;
   UP_DL_DAECHA_CLAMP.Visu_Adv_Arr[0] := FALSE;
   UP_DL_DAECHA_CLAMP.Visu_Adv_Arr[1] := FALSE;
   UP_DL_DAECHA_CLAMP.Visu_Adv_Arr[2] := FALSE;
   UP_DL_DAECHA_CLAMP.Visu_Adv_Arr[3] := FALSE;
   UP_DL_DAECHA_CLAMP.Visu_Adv_Arr[4] := FALSE;
   UP_DL_DAECHA_CLAMP.Visu_Adv_Arr[5] := FALSE;
   UP_DL_DAECHA_CLAMP.Visu_Adv_Arr[6] := FALSE;
   UP_DL_DAECHA_CLAMP.Visu_Adv_Arr[7] := FALSE;
   UP_DL_DAECHA_CLAMP.Visu_Adv_Arr[8] := FALSE;
   UP_DL_DAECHA_CLAMP.Visu_Adv_Arr[9] := FALSE;
   UP_DL_DAECHA_CLAMP.Visu_Adv_Arr[10] := FALSE;
   UP_DL_DAECHA_CLAMP.Visu_Adv_Arr[11] := FALSE;
   UP_DL_DAECHA_CLAMP.Visu_Adv_Arr[12] := FALSE;
   UP_DL_DAECHA_CLAMP.Visu_Adv_Arr[13] := FALSE;
   UP_DL_DAECHA_CLAMP.Visu_Adv_Arr[14] := FALSE;
   UP_DL_DAECHA_CLAMP.Visu_Adv_Arr[15] := FALSE;
   UP_DL_DAECHA_CLAMP.Visu_Ret_Arr[0] := TRUE;
   UP_DL_DAECHA_CLAMP.Visu_Ret_Arr[1] := TRUE;
   UP_DL_DAECHA_CLAMP.Visu_Ret_Arr[2] := TRUE;
   UP_DL_DAECHA_CLAMP.Visu_Ret_Arr[3] := FALSE;
   UP_DL_DAECHA_CLAMP.Visu_Ret_Arr[4] := FALSE;
   UP_DL_DAECHA_CLAMP.Visu_Ret_Arr[5] := FALSE;
   UP_DL_DAECHA_CLAMP.Visu_Ret_Arr[6] := FALSE;
   UP_DL_DAECHA_CLAMP.Visu_Ret_Arr[7] := FALSE;
   UP_DL_DAECHA_CLAMP.Visu_Ret_Arr[8] := FALSE;
   UP_DL_DAECHA_CLAMP.Visu_Ret_Arr[9] := FALSE;
   UP_DL_DAECHA_CLAMP.Visu_Ret_Arr[10] := FALSE;
   UP_DL_DAECHA_CLAMP.Visu_Ret_Arr[11] := FALSE;
   UP_DL_DAECHA_CLAMP.Visu_Ret_Arr[12] := FALSE;
   UP_DL_DAECHA_CLAMP.Visu_Ret_Arr[13] := FALSE;
   UP_DL_DAECHA_CLAMP.Visu_Ret_Arr[14] := FALSE;
   UP_DL_DAECHA_CLAMP.Visu_Ret_Arr[15] := FALSE;
   UP_DL_DAECHA_CLAMP.BLK_Move_Ret := 0;
   UP_DL_DAECHA_CLAMP.Enable := TRUE;
   UP_DL_DAECHA_CLAMP.Adv_End := FALSE;
   UP_DL_DAECHA_CLAMP.Ret_End := TRUE;
   UP_DL_AIR_ELE_UP_DOWN.Enable_Aux := TRUE;
   UP_DL_AIR_ELE_UP_DOWN.Adv_Amount := 1;
   UP_DL_AIR_ELE_UP_DOWN.Ret_Amount := 1;
   UP_DL_AIR_ELE_UP_DOWN.LS_Adv1 := FALSE;
   UP_DL_AIR_ELE_UP_DOWN.LS_Ret1 := TRUE;
   UP_DL_AIR_ELE_UP_DOWN.LS_Adv2 := FALSE;
   UP_DL_AIR_ELE_UP_DOWN.LS_Ret2 := FALSE;
   UP_DL_AIR_ELE_UP_DOWN.LS_Adv3 := FALSE;
   UP_DL_AIR_ELE_UP_DOWN.LS_Ret3 := FALSE;
   UP_DL_AIR_ELE_UP_DOWN.LS_Adv4 := FALSE;
   UP_DL_AIR_ELE_UP_DOWN.LS_Ret4 := FALSE;
   UP_DL_AIR_ELE_UP_DOWN.SOL_Adv := FALSE;
   UP_DL_AIR_ELE_UP_DOWN.SOL_Ret := FALSE;
   UP_DL_AIR_ELE_UP_DOWN.M_Ready := TRUE;
   UP_DL_AIR_ELE_UP_DOWN.T_CHK1 := T#4S;
   UP_DL_AIR_ELE_UP_DOWN.T_CHK2 := T#4S;
   UP_DL_AIR_ELE_UP_DOWN.PB_Lamp_CHK := FALSE;
   UP_DL_AIR_ELE_UP_DOWN.PB_Error_Rst := FALSE;
   UP_DL_AIR_ELE_UP_DOWN.M_FLICK := TRUE;
   UP_DL_AIR_ELE_UP_DOWN.M_Adv_Err := FALSE;
   UP_DL_AIR_ELE_UP_DOWN.M_Ret_Err := FALSE;
   UP_DL_AIR_ELE_UP_DOWN.LP_Adv := FALSE;
   UP_DL_AIR_ELE_UP_DOWN.LP_Ret := TRUE;
   UP_DL_AIR_ELE_UP_DOWN.Visu_Adv := W#16#0;
   UP_DL_AIR_ELE_UP_DOWN.Visu_Ret := W#16#300;
   UP_DL_AIR_ELE_UP_DOWN.Error_T1.IN := FALSE;
   UP_DL_AIR_ELE_UP_DOWN.Error_T1.PT := T#4S;
   UP_DL_AIR_ELE_UP_DOWN.Error_T1.Q := FALSE;
   UP_DL_AIR_ELE_UP_DOWN.Error_T1.ET := T#0MS;
   UP_DL_AIR_ELE_UP_DOWN.Error_T1.STATE := B#16#0;
   UP_DL_AIR_ELE_UP_DOWN.Error_T1.STIME := T#23D5H8M58S224MS;
   UP_DL_AIR_ELE_UP_DOWN.Error_T1.ATIME := T#23D5H8M58S774MS;
   UP_DL_AIR_ELE_UP_DOWN.Error_T2.IN := FALSE;
   UP_DL_AIR_ELE_UP_DOWN.Error_T2.PT := T#4S;
   UP_DL_AIR_ELE_UP_DOWN.Error_T2.Q := FALSE;
   UP_DL_AIR_ELE_UP_DOWN.Error_T2.ET := T#0MS;
   UP_DL_AIR_ELE_UP_DOWN.Error_T2.STATE := B#16#0;
   UP_DL_AIR_ELE_UP_DOWN.Error_T2.STIME := T#0MS;
   UP_DL_AIR_ELE_UP_DOWN.Error_T2.ATIME := T#0MS;
   UP_DL_AIR_ELE_UP_DOWN.CHK_Aux1 := FALSE;
   UP_DL_AIR_ELE_UP_DOWN.CHK_Aux2 := FALSE;
   UP_DL_AIR_ELE_UP_DOWN.Error_T1_DN := FALSE;
   UP_DL_AIR_ELE_UP_DOWN.Error_T2_DN := FALSE;
   UP_DL_AIR_ELE_UP_DOWN.Adv_Memo := FALSE;
   UP_DL_AIR_ELE_UP_DOWN.Visu_Adv_Arr[0] := FALSE;
   UP_DL_AIR_ELE_UP_DOWN.Visu_Adv_Arr[1] := FALSE;
   UP_DL_AIR_ELE_UP_DOWN.Visu_Adv_Arr[2] := FALSE;
   UP_DL_AIR_ELE_UP_DOWN.Visu_Adv_Arr[3] := FALSE;
   UP_DL_AIR_ELE_UP_DOWN.Visu_Adv_Arr[4] := FALSE;
   UP_DL_AIR_ELE_UP_DOWN.Visu_Adv_Arr[5] := FALSE;
   UP_DL_AIR_ELE_UP_DOWN.Visu_Adv_Arr[6] := FALSE;
   UP_DL_AIR_ELE_UP_DOWN.Visu_Adv_Arr[7] := FALSE;
   UP_DL_AIR_ELE_UP_DOWN.Visu_Adv_Arr[8] := FALSE;
   UP_DL_AIR_ELE_UP_DOWN.Visu_Adv_Arr[9] := FALSE;
   UP_DL_AIR_ELE_UP_DOWN.Visu_Adv_Arr[10] := FALSE;
   UP_DL_AIR_ELE_UP_DOWN.Visu_Adv_Arr[11] := FALSE;
   UP_DL_AIR_ELE_UP_DOWN.Visu_Adv_Arr[12] := FALSE;
   UP_DL_AIR_ELE_UP_DOWN.Visu_Adv_Arr[13] := FALSE;
   UP_DL_AIR_ELE_UP_DOWN.Visu_Adv_Arr[14] := FALSE;
   UP_DL_AIR_ELE_UP_DOWN.Visu_Adv_Arr[15] := FALSE;
   UP_DL_AIR_ELE_UP_DOWN.Visu_Ret_Arr[0] := TRUE;
   UP_DL_AIR_ELE_UP_DOWN.Visu_Ret_Arr[1] := TRUE;
   UP_DL_AIR_ELE_UP_DOWN.Visu_Ret_Arr[2] := FALSE;
   UP_DL_AIR_ELE_UP_DOWN.Visu_Ret_Arr[3] := FALSE;
   UP_DL_AIR_ELE_UP_DOWN.Visu_Ret_Arr[4] := FALSE;
   UP_DL_AIR_ELE_UP_DOWN.Visu_Ret_Arr[5] := FALSE;
   UP_DL_AIR_ELE_UP_DOWN.Visu_Ret_Arr[6] := FALSE;
   UP_DL_AIR_ELE_UP_DOWN.Visu_Ret_Arr[7] := FALSE;
   UP_DL_AIR_ELE_UP_DOWN.Visu_Ret_Arr[8] := FALSE;
   UP_DL_AIR_ELE_UP_DOWN.Visu_Ret_Arr[9] := FALSE;
   UP_DL_AIR_ELE_UP_DOWN.Visu_Ret_Arr[10] := FALSE;
   UP_DL_AIR_ELE_UP_DOWN.Visu_Ret_Arr[11] := FALSE;
   UP_DL_AIR_ELE_UP_DOWN.Visu_Ret_Arr[12] := FALSE;
   UP_DL_AIR_ELE_UP_DOWN.Visu_Ret_Arr[13] := FALSE;
   UP_DL_AIR_ELE_UP_DOWN.Visu_Ret_Arr[14] := FALSE;
   UP_DL_AIR_ELE_UP_DOWN.Visu_Ret_Arr[15] := FALSE;
   UP_DL_AIR_ELE_UP_DOWN.BLK_Move_Ret := 0;
   UP_DL_AIR_ELE_UP_DOWN.Enable := TRUE;
   UP_DL_AIR_ELE_UP_DOWN.Adv_End := FALSE;
   UP_DL_AIR_ELE_UP_DOWN.Ret_End := TRUE;
   UP_DL_AIR_ELE_ADV_RET.Enable_Aux := TRUE;
   UP_DL_AIR_ELE_ADV_RET.Adv_Amount := 1;
   UP_DL_AIR_ELE_ADV_RET.Ret_Amount := 1;
   UP_DL_AIR_ELE_ADV_RET.LS_Adv1 := FALSE;
   UP_DL_AIR_ELE_ADV_RET.LS_Ret1 := TRUE;
   UP_DL_AIR_ELE_ADV_RET.LS_Adv2 := FALSE;
   UP_DL_AIR_ELE_ADV_RET.LS_Ret2 := FALSE;
   UP_DL_AIR_ELE_ADV_RET.LS_Adv3 := FALSE;
   UP_DL_AIR_ELE_ADV_RET.LS_Ret3 := FALSE;
   UP_DL_AIR_ELE_ADV_RET.LS_Adv4 := FALSE;
   UP_DL_AIR_ELE_ADV_RET.LS_Ret4 := FALSE;
   UP_DL_AIR_ELE_ADV_RET.SOL_Adv := FALSE;
   UP_DL_AIR_ELE_ADV_RET.SOL_Ret := FALSE;
   UP_DL_AIR_ELE_ADV_RET.M_Ready := TRUE;
   UP_DL_AIR_ELE_ADV_RET.T_CHK1 := T#3S;
   UP_DL_AIR_ELE_ADV_RET.T_CHK2 := T#3S;
   UP_DL_AIR_ELE_ADV_RET.PB_Lamp_CHK := FALSE;
   UP_DL_AIR_ELE_ADV_RET.PB_Error_Rst := FALSE;
   UP_DL_AIR_ELE_ADV_RET.M_FLICK := TRUE;
   UP_DL_AIR_ELE_ADV_RET.M_Adv_Err := FALSE;
   UP_DL_AIR_ELE_ADV_RET.M_Ret_Err := FALSE;
   UP_DL_AIR_ELE_ADV_RET.LP_Adv := FALSE;
   UP_DL_AIR_ELE_ADV_RET.LP_Ret := TRUE;
   UP_DL_AIR_ELE_ADV_RET.Visu_Adv := W#16#0;
   UP_DL_AIR_ELE_ADV_RET.Visu_Ret := W#16#300;
   UP_DL_AIR_ELE_ADV_RET.Error_T1.IN := FALSE;
   UP_DL_AIR_ELE_ADV_RET.Error_T1.PT := T#3S;
   UP_DL_AIR_ELE_ADV_RET.Error_T1.Q := FALSE;
   UP_DL_AIR_ELE_ADV_RET.Error_T1.ET := T#0MS;
   UP_DL_AIR_ELE_ADV_RET.Error_T1.STATE := B#16#0;
   UP_DL_AIR_ELE_ADV_RET.Error_T1.STIME := T#23D5H8M58S22MS;
   UP_DL_AIR_ELE_ADV_RET.Error_T1.ATIME := T#23D5H8M58S202MS;
   UP_DL_AIR_ELE_ADV_RET.Error_T2.IN := FALSE;
   UP_DL_AIR_ELE_ADV_RET.Error_T2.PT := T#3S;
   UP_DL_AIR_ELE_ADV_RET.Error_T2.Q := FALSE;
   UP_DL_AIR_ELE_ADV_RET.Error_T2.ET := T#0MS;
   UP_DL_AIR_ELE_ADV_RET.Error_T2.STATE := B#16#0;
   UP_DL_AIR_ELE_ADV_RET.Error_T2.STIME := T#0MS;
   UP_DL_AIR_ELE_ADV_RET.Error_T2.ATIME := T#0MS;
   UP_DL_AIR_ELE_ADV_RET.CHK_Aux1 := FALSE;
   UP_DL_AIR_ELE_ADV_RET.CHK_Aux2 := FALSE;
   UP_DL_AIR_ELE_ADV_RET.Error_T1_DN := FALSE;
   UP_DL_AIR_ELE_ADV_RET.Error_T2_DN := FALSE;
   UP_DL_AIR_ELE_ADV_RET.Adv_Memo := FALSE;
   UP_DL_AIR_ELE_ADV_RET.Visu_Adv_Arr[0] := FALSE;
   UP_DL_AIR_ELE_ADV_RET.Visu_Adv_Arr[1] := FALSE;
   UP_DL_AIR_ELE_ADV_RET.Visu_Adv_Arr[2] := FALSE;
   UP_DL_AIR_ELE_ADV_RET.Visu_Adv_Arr[3] := FALSE;
   UP_DL_AIR_ELE_ADV_RET.Visu_Adv_Arr[4] := FALSE;
   UP_DL_AIR_ELE_ADV_RET.Visu_Adv_Arr[5] := FALSE;
   UP_DL_AIR_ELE_ADV_RET.Visu_Adv_Arr[6] := FALSE;
   UP_DL_AIR_ELE_ADV_RET.Visu_Adv_Arr[7] := FALSE;
   UP_DL_AIR_ELE_ADV_RET.Visu_Adv_Arr[8] := FALSE;
   UP_DL_AIR_ELE_ADV_RET.Visu_Adv_Arr[9] := FALSE;
   UP_DL_AIR_ELE_ADV_RET.Visu_Adv_Arr[10] := FALSE;
   UP_DL_AIR_ELE_ADV_RET.Visu_Adv_Arr[11] := FALSE;
   UP_DL_AIR_ELE_ADV_RET.Visu_Adv_Arr[12] := FALSE;
   UP_DL_AIR_ELE_ADV_RET.Visu_Adv_Arr[13] := FALSE;
   UP_DL_AIR_ELE_ADV_RET.Visu_Adv_Arr[14] := FALSE;
   UP_DL_AIR_ELE_ADV_RET.Visu_Adv_Arr[15] := FALSE;
   UP_DL_AIR_ELE_ADV_RET.Visu_Ret_Arr[0] := TRUE;
   UP_DL_AIR_ELE_ADV_RET.Visu_Ret_Arr[1] := TRUE;
   UP_DL_AIR_ELE_ADV_RET.Visu_Ret_Arr[2] := FALSE;
   UP_DL_AIR_ELE_ADV_RET.Visu_Ret_Arr[3] := FALSE;
   UP_DL_AIR_ELE_ADV_RET.Visu_Ret_Arr[4] := FALSE;
   UP_DL_AIR_ELE_ADV_RET.Visu_Ret_Arr[5] := FALSE;
   UP_DL_AIR_ELE_ADV_RET.Visu_Ret_Arr[6] := FALSE;
   UP_DL_AIR_ELE_ADV_RET.Visu_Ret_Arr[7] := FALSE;
   UP_DL_AIR_ELE_ADV_RET.Visu_Ret_Arr[8] := FALSE;
   UP_DL_AIR_ELE_ADV_RET.Visu_Ret_Arr[9] := FALSE;
   UP_DL_AIR_ELE_ADV_RET.Visu_Ret_Arr[10] := FALSE;
   UP_DL_AIR_ELE_ADV_RET.Visu_Ret_Arr[11] := FALSE;
   UP_DL_AIR_ELE_ADV_RET.Visu_Ret_Arr[12] := FALSE;
   UP_DL_AIR_ELE_ADV_RET.Visu_Ret_Arr[13] := FALSE;
   UP_DL_AIR_ELE_ADV_RET.Visu_Ret_Arr[14] := FALSE;
   UP_DL_AIR_ELE_ADV_RET.Visu_Ret_Arr[15] := FALSE;
   UP_DL_AIR_ELE_ADV_RET.BLK_Move_Ret := 0;
   UP_DL_AIR_ELE_ADV_RET.Enable := TRUE;
   UP_DL_AIR_ELE_ADV_RET.Adv_End := FALSE;
   UP_DL_AIR_ELE_ADV_RET.Ret_End := TRUE;
   UP_DL_LIFT_LOCK.Enable_Aux := TRUE;
   UP_DL_LIFT_LOCK.Adv_Amount := 2;
   UP_DL_LIFT_LOCK.Ret_Amount := 2;
   UP_DL_LIFT_LOCK.LS_Adv1 := FALSE;
   UP_DL_LIFT_LOCK.LS_Ret1 := TRUE;
   UP_DL_LIFT_LOCK.LS_Adv2 := FALSE;
   UP_DL_LIFT_LOCK.LS_Ret2 := TRUE;
   UP_DL_LIFT_LOCK.LS_Adv3 := FALSE;
   UP_DL_LIFT_LOCK.LS_Ret3 := FALSE;
   UP_DL_LIFT_LOCK.LS_Adv4 := FALSE;
   UP_DL_LIFT_LOCK.LS_Ret4 := FALSE;
   UP_DL_LIFT_LOCK.SOL_Adv := FALSE;
   UP_DL_LIFT_LOCK.SOL_Ret := FALSE;
   UP_DL_LIFT_LOCK.M_Ready := TRUE;
   UP_DL_LIFT_LOCK.T_CHK1 := T#5S;
   UP_DL_LIFT_LOCK.T_CHK2 := T#5S;
   UP_DL_LIFT_LOCK.PB_Lamp_CHK := FALSE;
   UP_DL_LIFT_LOCK.PB_Error_Rst := FALSE;
   UP_DL_LIFT_LOCK.M_FLICK := TRUE;
   UP_DL_LIFT_LOCK.M_Adv_Err := FALSE;
   UP_DL_LIFT_LOCK.M_Ret_Err := FALSE;
   UP_DL_LIFT_LOCK.LP_Adv := FALSE;
   UP_DL_LIFT_LOCK.LP_Ret := TRUE;
   UP_DL_LIFT_LOCK.Visu_Adv := W#16#0;
   UP_DL_LIFT_LOCK.Visu_Ret := W#16#700;
   UP_DL_LIFT_LOCK.Error_T1.IN := FALSE;
   UP_DL_LIFT_LOCK.Error_T1.PT := T#5S;
   UP_DL_LIFT_LOCK.Error_T1.Q := FALSE;
   UP_DL_LIFT_LOCK.Error_T1.ET := T#0MS;
   UP_DL_LIFT_LOCK.Error_T1.STATE := B#16#0;
   UP_DL_LIFT_LOCK.Error_T1.STIME := T#23D5H9M8S411MS;
   UP_DL_LIFT_LOCK.Error_T1.ATIME := T#23D5H9M9S401MS;
   UP_DL_LIFT_LOCK.Error_T2.IN := FALSE;
   UP_DL_LIFT_LOCK.Error_T2.PT := T#5S;
   UP_DL_LIFT_LOCK.Error_T2.Q := FALSE;
   UP_DL_LIFT_LOCK.Error_T2.ET := T#0MS;
   UP_DL_LIFT_LOCK.Error_T2.STATE := B#16#0;
   UP_DL_LIFT_LOCK.Error_T2.STIME := T#0MS;
   UP_DL_LIFT_LOCK.Error_T2.ATIME := T#0MS;
   UP_DL_LIFT_LOCK.CHK_Aux1 := FALSE;
   UP_DL_LIFT_LOCK.CHK_Aux2 := FALSE;
   UP_DL_LIFT_LOCK.Error_T1_DN := FALSE;
   UP_DL_LIFT_LOCK.Error_T2_DN := FALSE;
   UP_DL_LIFT_LOCK.Adv_Memo := FALSE;
   UP_DL_LIFT_LOCK.Visu_Adv_Arr[0] := FALSE;
   UP_DL_LIFT_LOCK.Visu_Adv_Arr[1] := FALSE;
   UP_DL_LIFT_LOCK.Visu_Adv_Arr[2] := FALSE;
   UP_DL_LIFT_LOCK.Visu_Adv_Arr[3] := FALSE;
   UP_DL_LIFT_LOCK.Visu_Adv_Arr[4] := FALSE;
   UP_DL_LIFT_LOCK.Visu_Adv_Arr[5] := FALSE;
   UP_DL_LIFT_LOCK.Visu_Adv_Arr[6] := FALSE;
   UP_DL_LIFT_LOCK.Visu_Adv_Arr[7] := FALSE;
   UP_DL_LIFT_LOCK.Visu_Adv_Arr[8] := FALSE;
   UP_DL_LIFT_LOCK.Visu_Adv_Arr[9] := FALSE;
   UP_DL_LIFT_LOCK.Visu_Adv_Arr[10] := FALSE;
   UP_DL_LIFT_LOCK.Visu_Adv_Arr[11] := FALSE;
   UP_DL_LIFT_LOCK.Visu_Adv_Arr[12] := FALSE;
   UP_DL_LIFT_LOCK.Visu_Adv_Arr[13] := FALSE;
   UP_DL_LIFT_LOCK.Visu_Adv_Arr[14] := FALSE;
   UP_DL_LIFT_LOCK.Visu_Adv_Arr[15] := FALSE;
   UP_DL_LIFT_LOCK.Visu_Ret_Arr[0] := TRUE;
   UP_DL_LIFT_LOCK.Visu_Ret_Arr[1] := TRUE;
   UP_DL_LIFT_LOCK.Visu_Ret_Arr[2] := TRUE;
   UP_DL_LIFT_LOCK.Visu_Ret_Arr[3] := FALSE;
   UP_DL_LIFT_LOCK.Visu_Ret_Arr[4] := FALSE;
   UP_DL_LIFT_LOCK.Visu_Ret_Arr[5] := FALSE;
   UP_DL_LIFT_LOCK.Visu_Ret_Arr[6] := FALSE;
   UP_DL_LIFT_LOCK.Visu_Ret_Arr[7] := FALSE;
   UP_DL_LIFT_LOCK.Visu_Ret_Arr[8] := FALSE;
   UP_DL_LIFT_LOCK.Visu_Ret_Arr[9] := FALSE;
   UP_DL_LIFT_LOCK.Visu_Ret_Arr[10] := FALSE;
   UP_DL_LIFT_LOCK.Visu_Ret_Arr[11] := FALSE;
   UP_DL_LIFT_LOCK.Visu_Ret_Arr[12] := FALSE;
   UP_DL_LIFT_LOCK.Visu_Ret_Arr[13] := FALSE;
   UP_DL_LIFT_LOCK.Visu_Ret_Arr[14] := FALSE;
   UP_DL_LIFT_LOCK.Visu_Ret_Arr[15] := FALSE;
   UP_DL_LIFT_LOCK.BLK_Move_Ret := 0;
   UP_DL_LIFT_LOCK.Enable := TRUE;
   UP_DL_LIFT_LOCK.Adv_End := FALSE;
   UP_DL_LIFT_LOCK.Ret_End := TRUE;
   UP_DL_LIFT.Enable_Aux := TRUE;
   UP_DL_LIFT.Adv_Amount := 1;
   UP_DL_LIFT.Ret_Amount := 1;
   UP_DL_LIFT.LS_Adv1 := FALSE;
   UP_DL_LIFT.LS_Ret1 := TRUE;
   UP_DL_LIFT.LS_Adv2 := FALSE;
   UP_DL_LIFT.LS_Ret2 := FALSE;
   UP_DL_LIFT.LS_Adv3 := FALSE;
   UP_DL_LIFT.LS_Ret3 := FALSE;
   UP_DL_LIFT.LS_Adv4 := FALSE;
   UP_DL_LIFT.LS_Ret4 := FALSE;
   UP_DL_LIFT.SOL_Adv := FALSE;
   UP_DL_LIFT.SOL_Ret := FALSE;
   UP_DL_LIFT.M_Ready := TRUE;
   UP_DL_LIFT.T_CHK1 := T#15S;
   UP_DL_LIFT.T_CHK2 := T#15S;
   UP_DL_LIFT.PB_Lamp_CHK := FALSE;
   UP_DL_LIFT.PB_Error_Rst := FALSE;
   UP_DL_LIFT.M_FLICK := TRUE;
   UP_DL_LIFT.M_Adv_Err := FALSE;
   UP_DL_LIFT.M_Ret_Err := FALSE;
   UP_DL_LIFT.LP_Adv := FALSE;
   UP_DL_LIFT.LP_Ret := TRUE;
   UP_DL_LIFT.Visu_Adv := W#16#0;
   UP_DL_LIFT.Visu_Ret := W#16#300;
   UP_DL_LIFT.Error_T1.IN := FALSE;
   UP_DL_LIFT.Error_T1.PT := T#15S;
   UP_DL_LIFT.Error_T1.Q := FALSE;
   UP_DL_LIFT.Error_T1.ET := T#0MS;
   UP_DL_LIFT.Error_T1.STATE := B#16#0;
   UP_DL_LIFT.Error_T1.STIME := T#23D5H9M9S932MS;
   UP_DL_LIFT.Error_T1.ATIME := T#23D5H9M17S645MS;
   UP_DL_LIFT.Error_T2.IN := FALSE;
   UP_DL_LIFT.Error_T2.PT := T#15S;
   UP_DL_LIFT.Error_T2.Q := FALSE;
   UP_DL_LIFT.Error_T2.ET := T#0MS;
   UP_DL_LIFT.Error_T2.STATE := B#16#0;
   UP_DL_LIFT.Error_T2.STIME := T#12D2H57M31S422MS;
   UP_DL_LIFT.Error_T2.ATIME := T#12D2H57M34S496MS;
   UP_DL_LIFT.CHK_Aux1 := FALSE;
   UP_DL_LIFT.CHK_Aux2 := FALSE;
   UP_DL_LIFT.Error_T1_DN := FALSE;
   UP_DL_LIFT.Error_T2_DN := FALSE;
   UP_DL_LIFT.Adv_Memo := FALSE;
   UP_DL_LIFT.Visu_Adv_Arr[0] := FALSE;
   UP_DL_LIFT.Visu_Adv_Arr[1] := FALSE;
   UP_DL_LIFT.Visu_Adv_Arr[2] := FALSE;
   UP_DL_LIFT.Visu_Adv_Arr[3] := FALSE;
   UP_DL_LIFT.Visu_Adv_Arr[4] := FALSE;
   UP_DL_LIFT.Visu_Adv_Arr[5] := FALSE;
   UP_DL_LIFT.Visu_Adv_Arr[6] := FALSE;
   UP_DL_LIFT.Visu_Adv_Arr[7] := FALSE;
   UP_DL_LIFT.Visu_Adv_Arr[8] := FALSE;
   UP_DL_LIFT.Visu_Adv_Arr[9] := FALSE;
   UP_DL_LIFT.Visu_Adv_Arr[10] := FALSE;
   UP_DL_LIFT.Visu_Adv_Arr[11] := FALSE;
   UP_DL_LIFT.Visu_Adv_Arr[12] := FALSE;
   UP_DL_LIFT.Visu_Adv_Arr[13] := FALSE;
   UP_DL_LIFT.Visu_Adv_Arr[14] := FALSE;
   UP_DL_LIFT.Visu_Adv_Arr[15] := FALSE;
   UP_DL_LIFT.Visu_Ret_Arr[0] := TRUE;
   UP_DL_LIFT.Visu_Ret_Arr[1] := TRUE;
   UP_DL_LIFT.Visu_Ret_Arr[2] := FALSE;
   UP_DL_LIFT.Visu_Ret_Arr[3] := FALSE;
   UP_DL_LIFT.Visu_Ret_Arr[4] := FALSE;
   UP_DL_LIFT.Visu_Ret_Arr[5] := FALSE;
   UP_DL_LIFT.Visu_Ret_Arr[6] := FALSE;
   UP_DL_LIFT.Visu_Ret_Arr[7] := FALSE;
   UP_DL_LIFT.Visu_Ret_Arr[8] := FALSE;
   UP_DL_LIFT.Visu_Ret_Arr[9] := FALSE;
   UP_DL_LIFT.Visu_Ret_Arr[10] := FALSE;
   UP_DL_LIFT.Visu_Ret_Arr[11] := FALSE;
   UP_DL_LIFT.Visu_Ret_Arr[12] := FALSE;
   UP_DL_LIFT.Visu_Ret_Arr[13] := FALSE;
   UP_DL_LIFT.Visu_Ret_Arr[14] := FALSE;
   UP_DL_LIFT.Visu_Ret_Arr[15] := FALSE;
   UP_DL_LIFT.BLK_Move_Ret := 0;
   UP_DL_LIFT.Enable := TRUE;
   UP_DL_LIFT.Adv_End := FALSE;
   UP_DL_LIFT.Ret_End := TRUE;
END_DATA_BLOCK

FUNCTION FC 151 : VOID
TITLE =
VERSION : 0.1

BEGIN
NETWORK
TITLE =
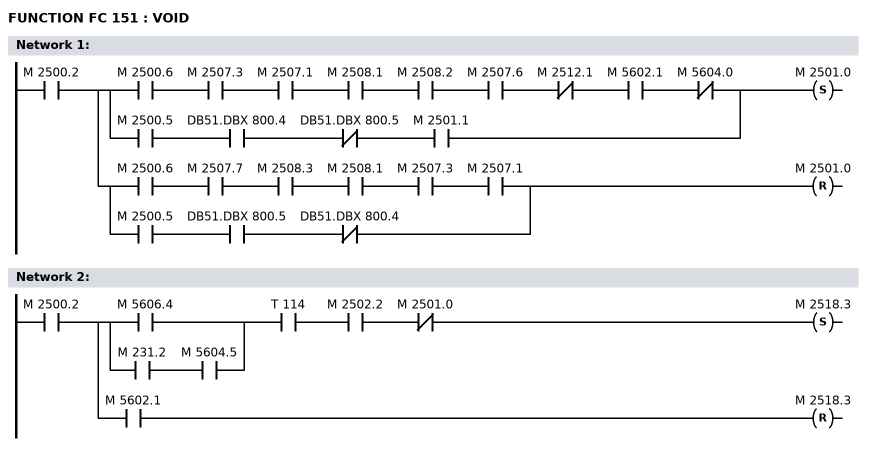

      A     M   2500.2;
      =     L      0.0;
      A     L      0.0;
      A(    ;
      A     M   2500.6;
      A     M   2507.3;
      A     M   2507.1;
      A     M   2508.1;
      A     M   2508.2;
      A     M   2507.6;
      AN    M   2512.1;
      A     M   5602.1;
      AN    M   5604.0;
      O     ;
      A     M   2500.5;
      A     DB51.DBX  800.4;
      AN    DB51.DBX  800.5;
      A     M   2501.1;
      )     ;
      S     M   2501.0;
      A     L      0.0;
      A(    ;
      A     M   2500.6;
      A     M   2507.7;
      A     M   2508.3;
      A     M   2508.1;
      A     M   2507.3;
      A     M   2507.1;
      O     ;
      A     M   2500.5;
      A     DB51.DBX  800.5;
      AN    DB51.DBX  800.4;
      )     ;
      R     M   2501.0;
NETWORK
TITLE =

      A     M   2500.2;
      =     L      0.0;
      A     L      0.0;
      A(    ;
      O     M   5606.4;
      O     ;
      A     M    231.2;
      A     M   5604.5;
      )     ;
      A     T    114;
      A     M   2502.2;
      AN    M   2501.0;
      S     M   2518.3;
      A     L      0.0;
      A     M   5602.1;
      R     M   2518.3;
END_FUNCTION

FUNCTION_BLOCK FB 152
TITLE =
VERSION : 0.1

BEGIN
NETWORK
TITLE =

      AN    OV;
      =     L      0.0;
      A     L      0.0;
      A     M   2500.6;
      A(    ;
      O     M    224.1;
      O     M    224.0;
      )     ;
      A     M   2005.4;
      A(    ;
      O     I    121.3;
      O     ;
      A     M    224.0;
      A     M   2005.4;
      )     ;
      S     M   2506.0;
      A     L      0.0;
      A     M   2506.0;
      A     M   2518.3;
      R     M   2506.0;
      A     L      0.0;
      A     M   2500.6;
      A(    ;
      O     M    224.1;
      O     ;
      A     M    224.0;
      AN    M      3.3;
      )     ;
      A     M   2005.4;
      A     M   2507.7;
      AN    M   2509.0;
      AN    I    121.3;
      AN    M      3.3;
      AN    M   2504.0;
      AN    M   2504.1;
      AN    M   2504.2;
      S     M   2506.1;
      A     L      0.0;
      A     M   2506.1;
      A     I    121.3;
      A     I     80.1;
      R     M   2506.1;
NETWORK
TITLE =
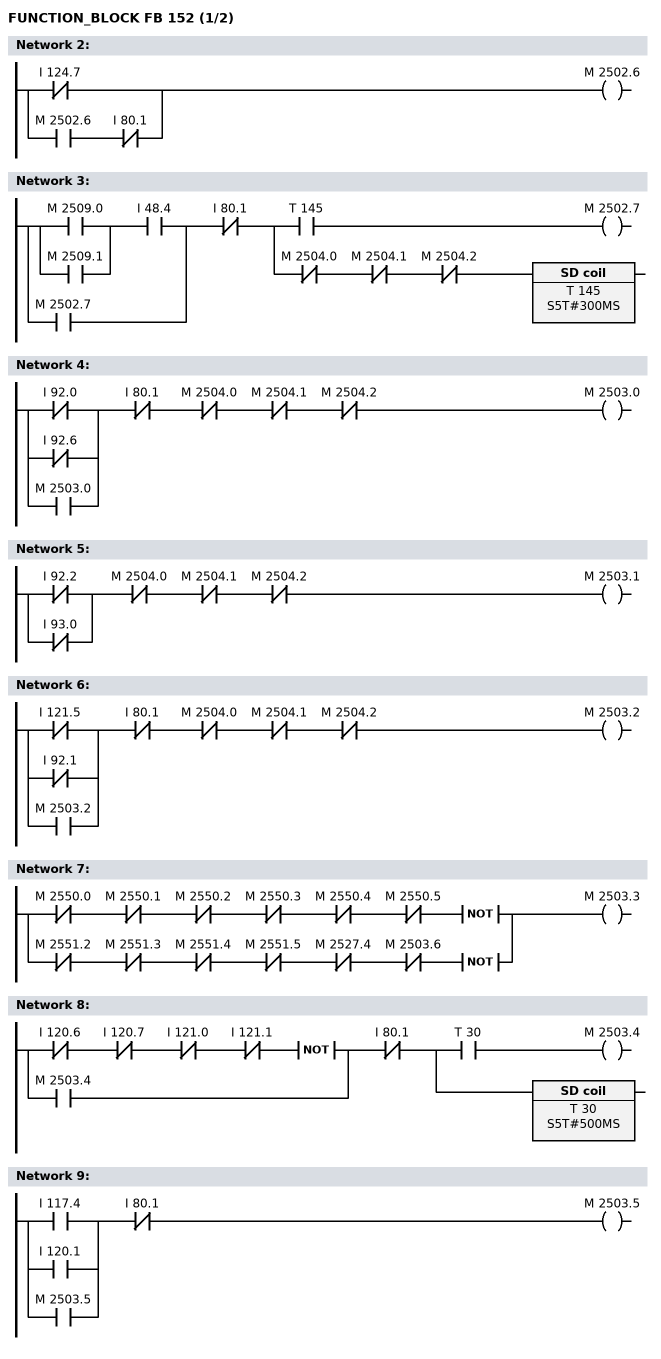

      ON    I    124.7;
      O     ;
      A     M   2502.6;
      AN    I     80.1;
      =     M   2502.6;
NETWORK
TITLE =

      A(    ;
      A(    ;
      O     M   2509.0;
      O     M   2509.1;
      )     ;
      A     I     48.4;
      O     M   2502.7;
      )     ;
      AN    I     80.1;
      =     L      0.0;
      A     L      0.0;
      A     T    145;
      =     M   2502.7;
      A     L      0.0;
      AN    M   2504.0;
      AN    M   2504.1;
      AN    M   2504.2;
      L     S5T#300MS;
      SD    T    145;
NETWORK
TITLE =

      A(    ;
      ON    I     92.0;
      ON    I     92.6;
      O     M   2503.0;
      )     ;
      AN    I     80.1;
      AN    M   2504.0;
      AN    M   2504.1;
      AN    M   2504.2;
      =     M   2503.0;
NETWORK
TITLE =

      A(    ;
      ON    I     92.2;
      ON    I     93.0;
      )     ;
      AN    M   2504.0;
      AN    M   2504.1;
      AN    M   2504.2;
      =     M   2503.1;
NETWORK
TITLE =

      A(    ;
      ON    I    121.5;
      ON    I     92.1;
      O     M   2503.2;
      )     ;
      AN    I     80.1;
      AN    M   2504.0;
      AN    M   2504.1;
      AN    M   2504.2;
      =     M   2503.2;
NETWORK
TITLE =

      AN    M   2550.0;
      AN    M   2550.1;
      AN    M   2550.2;
      AN    M   2550.3;
      AN    M   2550.4;
      AN    M   2550.5;
      NOT   ;
      O(    ;
      AN    M   2551.2;
      AN    M   2551.3;
      AN    M   2551.4;
      AN    M   2551.5;
      AN    M   2527.4;
      AN    M   2503.6;
      NOT   ;
      )     ;
      =     M   2503.3;
NETWORK
TITLE =

      A(    ;
      AN    I    120.6;
      AN    I    120.7;
      AN    I    121.0;
      AN    I    121.1;
      NOT   ;
      O     M   2503.4;
      )     ;
      AN    I     80.1;
      =     L      0.0;
      A     L      0.0;
      A     T     30;
      =     M   2503.4;
      A     L      0.0;
      BLD   102;
      L     S5T#500MS;
      SD    T     30;
NETWORK
TITLE =

      A(    ;
      O     I    117.4;
      O     I    120.1;
      O     M   2503.5;
      )     ;
      AN    I     80.1;
      =     M   2503.5;
NETWORK
TITLE =
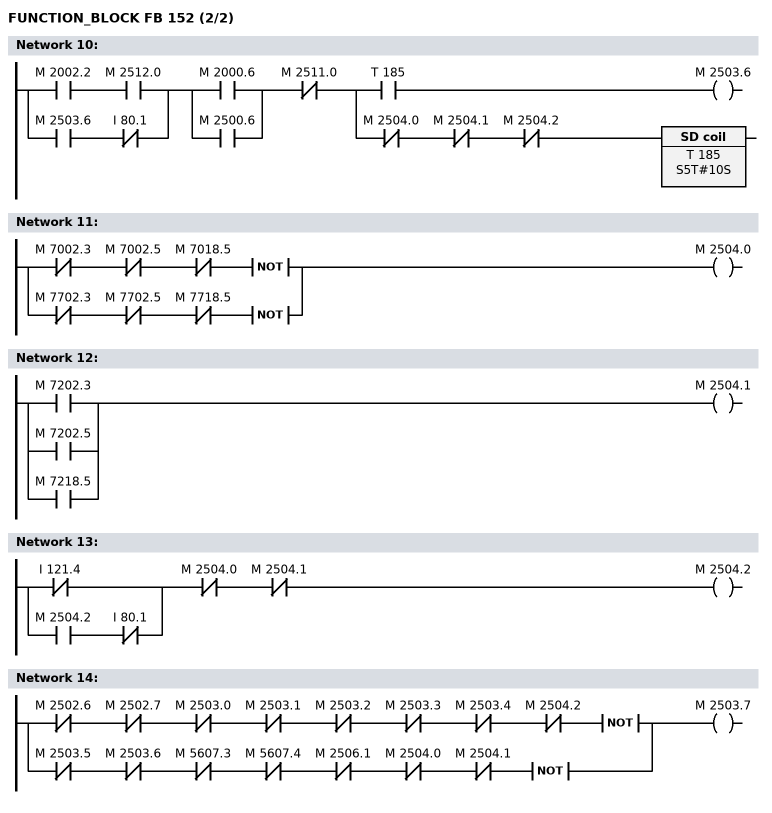

      A(    ;
      A     M   2002.2;
      A     M   2512.0;
      O     ;
      A     M   2503.6;
      AN    I     80.1;
      )     ;
      A(    ;
      O     M   2000.6;
      O     M   2500.6;
      )     ;
      AN    M   2511.0;
      =     L      0.0;
      A     L      0.0;
      A     T    185;
      =     M   2503.6;
      A     L      0.0;
      AN    M   2504.0;
      AN    M   2504.1;
      AN    M   2504.2;
      L     S5T#10S;
      SD    T    185;
NETWORK
TITLE =

      AN    M   7002.3;
      AN    M   7002.5;
      AN    M   7018.5;
      NOT   ;
      O(    ;
      AN    M   7702.3;
      AN    M   7702.5;
      AN    M   7718.5;
      NOT   ;
      )     ;
      =     M   2504.0;
NETWORK
TITLE =

      O     M   7202.3;
      O     M   7202.5;
      O     M   7218.5;
      =     M   2504.1;
NETWORK
TITLE =

      A(    ;
      ON    I    121.4;
      O     ;
      A     M   2504.2;
      AN    I     80.1;
      )     ;
      AN    M   2504.0;
      AN    M   2504.1;
      =     M   2504.2;
NETWORK
TITLE =

      AN    M   2502.6;
      AN    M   2502.7;
      AN    M   2503.0;
      AN    M   2503.1;
      AN    M   2503.2;
      AN    M   2503.3;
      AN    M   2503.4;
      AN    M   2504.2;
      NOT   ;
      O(    ;
      AN    M   2503.5;
      AN    M   2503.6;
      AN    M   5607.3;
      AN    M   5607.4;
      AN    M   2506.1;
      AN    M   2504.0;
      AN    M   2504.1;
      NOT   ;
      )     ;
      =     M   2503.7;
END_FUNCTION_BLOCK

DATA_BLOCK DB 152
TITLE =
VERSION : 0.0

 FB 152
BEGIN
END_DATA_BLOCK

FUNCTION FC 152 : VOID
TITLE =
VERSION : 0.1

BEGIN
NETWORK
TITLE =
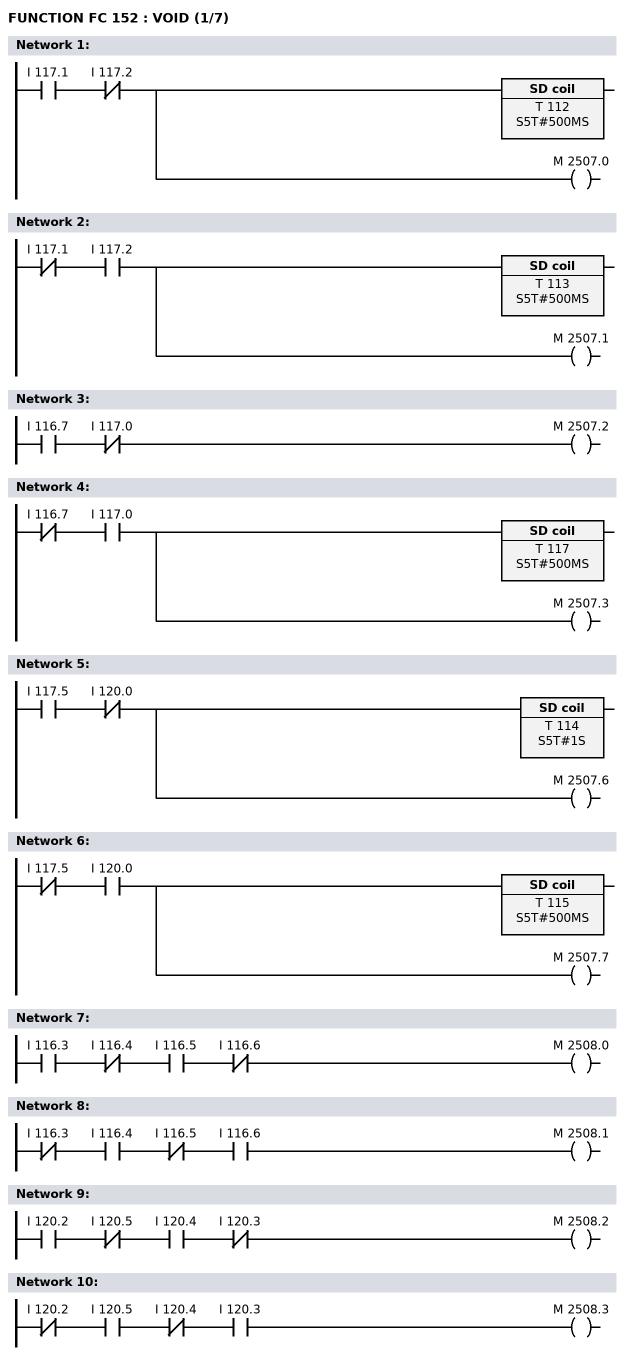

      A     I    117.1;
      AN    I    117.2;
      L     S5T#500MS;
      SD    T    112;
      =     M   2507.0;
NETWORK
TITLE =

      AN    I    117.1;
      A     I    117.2;
      L     S5T#500MS;
      SD    T    113;
      =     M   2507.1;
NETWORK
TITLE =

      A     I    116.7;
      AN    I    117.0;
      =     M   2507.2;
NETWORK
TITLE =

      AN    I    116.7;
      A     I    117.0;
      L     S5T#500MS;
      SD    T    117;
      =     M   2507.3;
NETWORK
TITLE =

      A     I    117.5;
      AN    I    120.0;
      L     S5T#1S;
      SD    T    114;
      =     M   2507.6;
NETWORK
TITLE =

      AN    I    117.5;
      A     I    120.0;
      L     S5T#500MS;
      SD    T    115;
      =     M   2507.7;
NETWORK
TITLE =

      A     I    116.3;
      AN    I    116.4;
      A     I    116.5;
      AN    I    116.6;
      =     M   2508.0;
NETWORK
TITLE =

      AN    I    116.3;
      A     I    116.4;
      AN    I    116.5;
      A     I    116.6;
      =     M   2508.1;
NETWORK
TITLE =

      A     I    120.2;
      AN    I    120.5;
      A     I    120.4;
      AN    I    120.3;
      =     M   2508.2;
NETWORK
TITLE =

      AN    I    120.2;
      A     I    120.5;
      AN    I    120.4;
      A     I    120.3;
      =     M   2508.3;
NETWORK
TITLE =
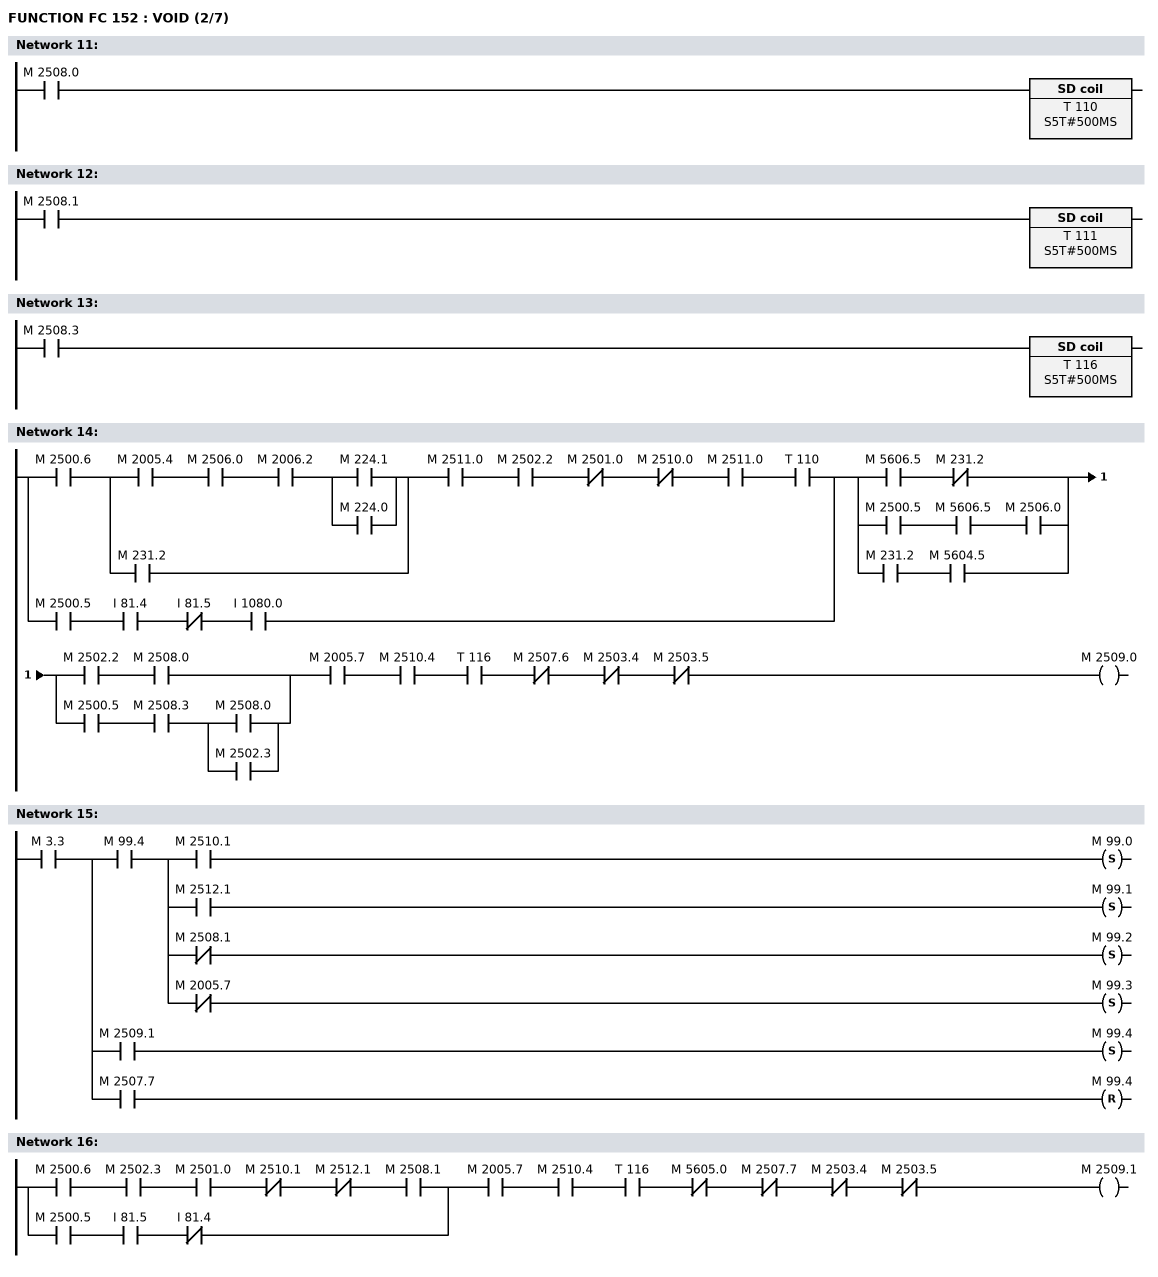

      A     M   2508.0;
      L     S5T#500MS;
      SD    T    110;
NETWORK
TITLE =

      A     M   2508.1;
      L     S5T#500MS;
      SD    T    111;
NETWORK
TITLE =

      A     M   2508.3;
      L     S5T#500MS;
      SD    T    116;
NETWORK
TITLE =

      A(    ;
      A     M   2500.6;
      A(    ;
      A     M   2005.4;
      A     M   2506.0;
      A     M   2006.2;
      A(    ;
      O     M    224.1;
      O     M    224.0;
      )     ;
      O     M    231.2;
      )     ;
      A     M   2511.0;
      A     M   2502.2;
      AN    M   2501.0;
      AN    M   2510.0;
      A     M   2511.0;
      A     T    110;
      O     ;
      A     M   2500.5;
      A     I     81.4;
      AN    I     81.5;
      A     I   1080.0;
      )     ;
      A(    ;
      A     M   5606.5;
      AN    M    231.2;
      O     ;
      A     M   2500.5;
      A     M   5606.5;
      A     M   2506.0;
      O     ;
      A     M    231.2;
      A     M   5604.5;
      )     ;
      A(    ;
      A     M   2502.2;
      A     M   2508.0;
      O     ;
      A     M   2500.5;
      A     M   2508.3;
      A(    ;
      O     M   2508.0;
      O     M   2502.3;
      )     ;
      )     ;
      A     M   2005.7;
      A     M   2510.4;
      A     T    116;
      AN    M   2507.6;
      AN    M   2503.4;
      AN    M   2503.5;
      =     M   2509.0;
NETWORK
TITLE =

      A     M      3.3;
      =     L      0.0;
      A     L      0.0;
      A     M     99.4;
      =     L      0.1;
      A     L      0.1;
      A     M   2510.1;
      S     M     99.0;
      A     L      0.1;
      A     M   2512.1;
      S     M     99.1;
      A     L      0.1;
      AN    M   2508.1;
      S     M     99.2;
      A     L      0.1;
      AN    M   2005.7;
      S     M     99.3;
      A     L      0.0;
      A     M   2509.1;
      S     M     99.4;
      A     L      0.0;
      A     M   2507.7;
      R     M     99.4;
NETWORK
TITLE =

      A(    ;
      A     M   2500.6;
      A     M   2502.3;
      A     M   2501.0;
      AN    M   2510.1;
      AN    M   2512.1;
      A     M   2508.1;
      O     ;
      A     M   2500.5;
      A     I     81.5;
      AN    I     81.4;
      )     ;
      A     M   2005.7;
      A     M   2510.4;
      A     T    116;
      AN    M   5605.0;
      AN    M   2507.7;
      AN    M   2503.4;
      AN    M   2503.5;
      =     M   2509.1;
NETWORK
TITLE =
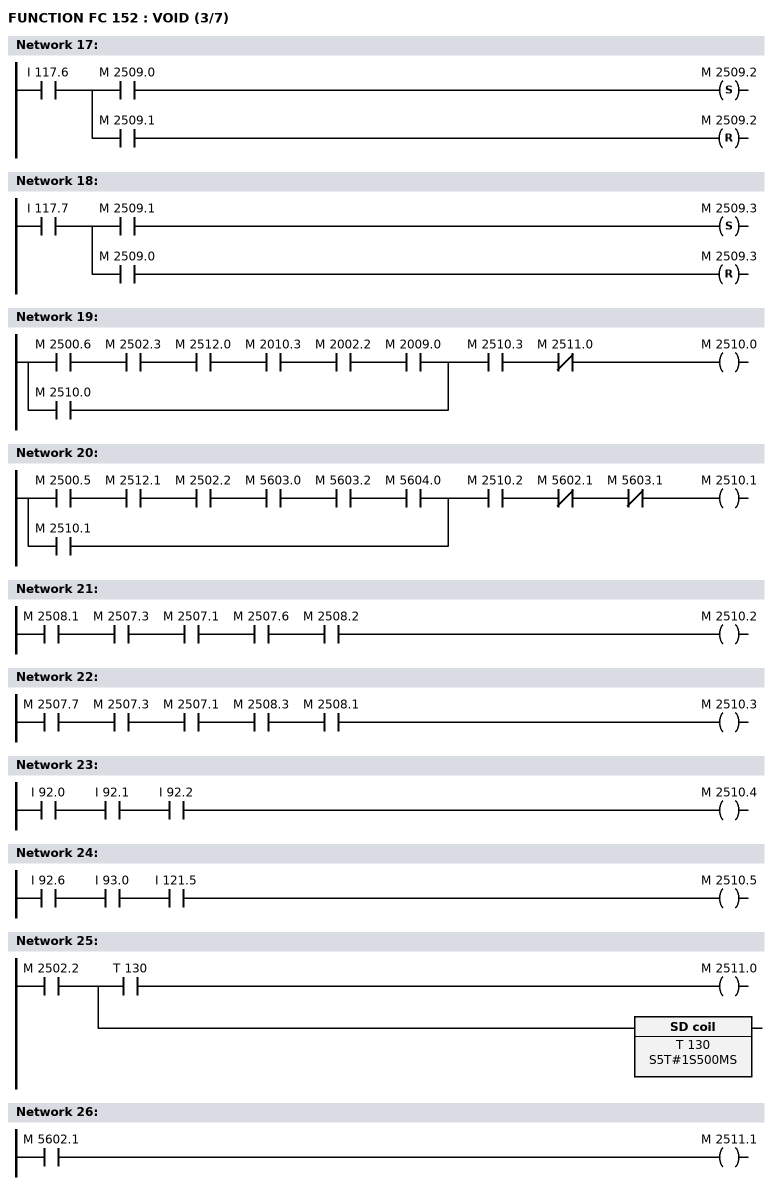

      A     I    117.6;
      =     L      0.0;
      A     L      0.0;
      A     M   2509.0;
      S     M   2509.2;
      A     L      0.0;
      A     M   2509.1;
      R     M   2509.2;
NETWORK
TITLE =

      A     I    117.7;
      =     L      0.0;
      A     L      0.0;
      A     M   2509.1;
      S     M   2509.3;
      A     L      0.0;
      A     M   2509.0;
      R     M   2509.3;
NETWORK
TITLE =

      A(    ;
      A     M   2500.6;
      A     M   2502.3;
      A     M   2512.0;
      A     M   2010.3;
      A     M   2002.2;
      A     M   2009.0;
      O     M   2510.0;
      )     ;
      A     M   2510.3;
      AN    M   2511.0;
      =     M   2510.0;
NETWORK
TITLE =

      A(    ;
      A     M   2500.5;
      A     M   2512.1;
      A     M   2502.2;
      A     M   5603.0;
      A     M   5603.2;
      A     M   5604.0;
      O     M   2510.1;
      )     ;
      A     M   2510.2;
      AN    M   5602.1;
      AN    M   5603.1;
      =     M   2510.1;
NETWORK
TITLE =

      A     M   2508.1;
      A     M   2507.3;
      A     M   2507.1;
      A     M   2507.6;
      A     M   2508.2;
      =     M   2510.2;
NETWORK
TITLE =

      A     M   2507.7;
      A     M   2507.3;
      A     M   2507.1;
      A     M   2508.3;
      A     M   2508.1;
      =     M   2510.3;
NETWORK
TITLE =

      A     I     92.0;
      A     I     92.1;
      A     I     92.2;
      =     M   2510.4;
NETWORK
TITLE =

      A     I     92.6;
      A     I     93.0;
      A     I    121.5;
      =     M   2510.5;
NETWORK
TITLE =

      A     M   2502.2;
      =     L      0.0;
      A     L      0.0;
      A     T    130;
      =     M   2511.0;
      A     L      0.0;
      BLD   102;
      L     S5T#1S500MS;
      SD    T    130;
NETWORK
TITLE =

      A     M   5602.1;
      =     M   2511.1;
NETWORK
TITLE =
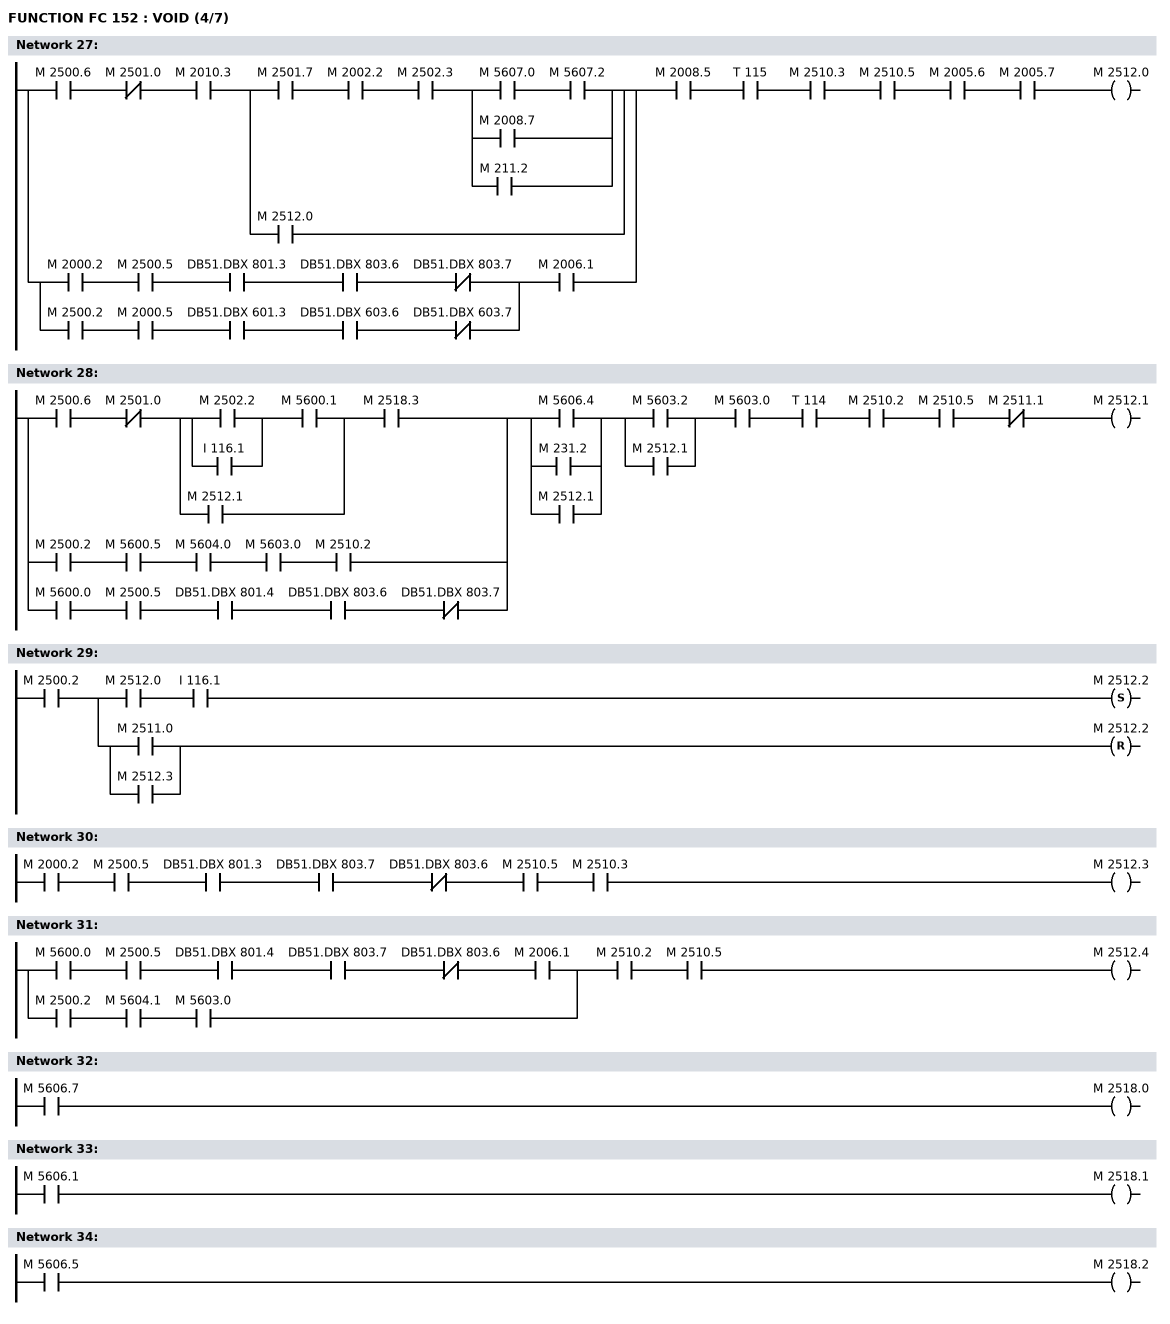

      A(    ;
      A     M   2500.6;
      AN    M   2501.0;
      A     M   2010.3;
      A(    ;
      A     M   2501.7;
      A     M   2002.2;
      A     M   2502.3;
      A(    ;
      A     M   5607.0;
      A     M   5607.2;
      O     M   2008.7;
      O     M    211.2;
      )     ;
      O     M   2512.0;
      )     ;
      O     ;
      A(    ;
      A     M   2000.2;
      A     M   2500.5;
      A     DB51.DBX  801.3;
      A     DB51.DBX  803.6;
      AN    DB51.DBX  803.7;
      O     ;
      A     M   2500.2;
      A     M   2000.5;
      A     DB51.DBX  601.3;
      A     DB51.DBX  603.6;
      AN    DB51.DBX  603.7;
      )     ;
      A     M   2006.1;
      )     ;
      A     M   2008.5;
      A     T    115;
      A     M   2510.3;
      A     M   2510.5;
      A     M   2005.6;
      A     M   2005.7;
      =     M   2512.0;
NETWORK
TITLE =

      A(    ;
      A     M   2500.6;
      AN    M   2501.0;
      A(    ;
      A(    ;
      O     M   2502.2;
      O     I    116.1;
      )     ;
      A     M   5600.1;
      O     M   2512.1;
      )     ;
      A     M   2518.3;
      O     ;
      A     M   2500.2;
      A     M   5600.5;
      A     M   5604.0;
      A     M   5603.0;
      A     M   2510.2;
      O     ;
      A     M   5600.0;
      A     M   2500.5;
      A     DB51.DBX  801.4;
      A     DB51.DBX  803.6;
      AN    DB51.DBX  803.7;
      )     ;
      A(    ;
      O     M   5606.4;
      O     M    231.2;
      O     M   2512.1;
      )     ;
      A(    ;
      O     M   5603.2;
      O     M   2512.1;
      )     ;
      A     M   5603.0;
      A     T    114;
      A     M   2510.2;
      A     M   2510.5;
      AN    M   2511.1;
      =     M   2512.1;
NETWORK
TITLE =

      A     M   2500.2;
      =     L      0.0;
      A     L      0.0;
      A     M   2512.0;
      A     I    116.1;
      S     M   2512.2;
      A     L      0.0;
      A(    ;
      O     M   2511.0;
      O     M   2512.3;
      )     ;
      R     M   2512.2;
NETWORK
TITLE =

      A     M   2000.2;
      A     M   2500.5;
      A     DB51.DBX  801.3;
      A     DB51.DBX  803.7;
      AN    DB51.DBX  803.6;
      A     M   2510.5;
      A     M   2510.3;
      =     M   2512.3;
NETWORK
TITLE =

      A(    ;
      A     M   5600.0;
      A     M   2500.5;
      A     DB51.DBX  801.4;
      A     DB51.DBX  803.7;
      AN    DB51.DBX  803.6;
      A     M   2006.1;
      O     ;
      A     M   2500.2;
      A     M   5604.1;
      A     M   5603.0;
      )     ;
      A     M   2510.2;
      A     M   2510.5;
      =     M   2512.4;
NETWORK
TITLE =

      A     M   5606.7;
      =     M   2518.0;
NETWORK
TITLE =

      A     M   5606.1;
      =     M   2518.1;
NETWORK
TITLE =

      A     M   5606.5;
      =     M   2518.2;
NETWORK
TITLE =
